// TwinCAT 3 PLC project mobject_core
// Title: mobject-core
// Company: mobject
// Author: mobject dev team
// ProjectVersion: 0.4.0
// ProgramVersion: 3.1.4024.0
// libraries:
//   Tc2_Standard, * (Beckhoff Automation GmbH)
//   Tc2_System, * (Beckhoff Automation GmbH)
//   Tc2_Utilities, * (Beckhoff Automation GmbH)
//   Tc3_DynamicMemory, * (Beckhoff Automation GmbH)
//   Tc3_JsonXml, * (Beckhoff Automation GmbH)
// project tree:
//   mobject-collections/Dictionary/ Dictionary.TcPOU
//   mobject-collections/Interfaces/Collections/Events/ I_CollectionChangedEvent.TcIO (not stored), I_CollectionDisposedEvent.TcIO (not stored)
//   mobject-collections/Interfaces/Collections/ I_Collection.TcIO, I_LinkedList.TcIO, I_List.TcIO (not stored), I_Queue.TcIO (not stored), I_Stack.TcIO
//   mobject-collections/Interfaces/Collections/Nodes/ I_CollectionNode.TcIO (not stored), I_LinkedListNode.TcIO (not stored), I_ListNode.TcIO (not stored)
//   mobject-collections/Interfaces/KeyValueCollections/Events/ I_KeyValueCollectionChangedEvent.TcIO (not stored), I_KeyValueCollectionDisposedEvent.TcIO (not stored)
//   mobject-collections/Interfaces/KeyValueCollections/ I_Dictionary.TcIO (not stored), I_KeyValueCollection.TcIO (not stored)
//   mobject-collections/Interfaces/KeyValueCollections/Nodes/ I_DictionaryTreeNode.TcIO, I_OrderedDictionaryTreeNode.TcIO
//   mobject-collections/LinkedList/ LinkedList.TcPOU
//   mobject-collections/List/ List.TcPOU
//   mobject-collections/OrderedDictionary/ OrderedDictionary.TcPOU
//   mobject-collections/Queue/ Queue.TcPOU (not stored)
//   mobject-collections/Stack/ Stack.TcPOU
//   mobject-collections/_Internal/Dictionary/Enumerator/ DictionaryForwardEnumerator.TcPOU
//   mobject-collections/_Internal/Dictionary/Node/ DictionaryTreeNode.TcPOU
//   mobject-collections/_Internal/Events/Collection/ CollectionChangedEvent.TcPOU (not stored), CollectionDisposedEvent.TcPOU (not stored), CollectionEvent.TcPOU (not stored)
//   mobject-collections/_Internal/Events/KeyValueCollection/ KeyValueCollectionChangedEvent.TcPOU, KeyValueCollectionDisposedEvent.TcPOU, KeyValueCollectionEvent.TcPOU
//   mobject-collections/_Internal/LinkedList/Enumerator/ LinkedListForwardEnumerator.TcPOU
//   mobject-collections/_Internal/LinkedList/Node/ LinkedListNode.TcPOU
//   mobject-collections/_Internal/List/Node/ ListNode.TcPOU
//   mobject-collections/_Internal/OrderedDictionary/Enumerator/ OrderedDictionaryForwardEnumerator.TcPOU (not stored)
//   mobject-collections/_Internal/OrderedDictionary/Node/ OrderedDictionaryTreeNode.TcPOU
//   mobject-commands/AsyncCommand/ AsyncCommand.TcPOU (not stored)
//   mobject-commands/AsyncCommand/Interface/ I_AsyncCommand.TcIO
//   mobject-commands/AsyncCommand/Runners/ SingleAsyncCommandRunner.TcPOU (not stored)
//   mobject-commands/Command/Interface/ I_Command.TcIO
//   mobject-commands/_Internal/AsyncCommandStateMachine/ AsyncCommandStateMachine.TcPOU, I_AsyncCommandStateControl.TcIO (not stored)
//   mobject-constants/ DatatypeLimits.TcGVL
//   mobject-converters/Converters/BOOL_TO_/ TryConvert_BOOL_TO_BOOL.TcPOU (not stored), TryConvert_BOOL_TO_BYTE.TcPOU, TryConvert_BOOL_TO_DATE.TcPOU, TryConvert_BOOL_TO_Destination.TcPOU, TryConvert_BOOL_TO_DINT.TcPOU, TryConvert_BOOL_TO_DT.TcPOU (not stored), TryConvert_BOOL_TO_DWORD.TcPOU (not stored), TryConvert_BOOL_TO_INT.TcPOU, TryConvert_BOOL_TO_LINT.TcPOU, TryConvert_BOOL_TO_LREAL.TcPOU (not stored), TryConvert_BOOL_TO_LWORD.TcPOU (not stored), TryConvert_BOOL_TO_REAL.TcPOU, TryConvert_BOOL_TO_SINT.TcPOU (not stored), TryConvert_BOOL_TO_STRING.TcPOU (not stored), TryConvert_BOOL_TO_TIME.TcPOU (not stored), TryConvert_BOOL_TO_TOD.TcPOU (not stored), TryConvert_BOOL_TO_UDINT.TcPOU, TryConvert_BOOL_TO_UINT.TcPOU, TryConvert_BOOL_TO_ULINT.TcPOU, TryConvert_BOOL_TO_USINT.TcPOU, TryConvert_BOOL_TO_WORD.TcPOU (not stored)
//   mobject-converters/Converters/BYTE_TO_/ TryConvert_BYTE_TO_BOOL.TcPOU, TryConvert_BYTE_TO_BYTE.TcPOU (not stored), TryConvert_BYTE_TO_DATE.TcPOU, TryConvert_BYTE_TO_Destination.TcPOU (not stored), TryConvert_BYTE_TO_DINT.TcPOU, TryConvert_BYTE_TO_DT.TcPOU (not stored), TryConvert_BYTE_TO_DWORD.TcPOU, TryConvert_BYTE_TO_INT.TcPOU, TryConvert_BYTE_TO_LINT.TcPOU (not stored), TryConvert_BYTE_TO_LREAL.TcPOU (not stored), TryConvert_BYTE_TO_LWORD.TcPOU (not stored), TryConvert_BYTE_TO_REAL.TcPOU, TryConvert_BYTE_TO_SINT.TcPOU, TryConvert_BYTE_TO_STRING.TcPOU, TryConvert_BYTE_TO_TIME.TcPOU, TryConvert_BYTE_TO_TOD.TcPOU, TryConvert_BYTE_TO_UDINT.TcPOU (not stored), TryConvert_BYTE_TO_UINT.TcPOU (not stored), TryConvert_BYTE_TO_ULINT.TcPOU, TryConvert_BYTE_TO_USINT.TcPOU, TryConvert_BYTE_TO_WORD.TcPOU
//   mobject-converters/Converters/DATE_TO_/ TryConvert_DATE_TO_BOOL.TcPOU (not stored), TryConvert_DATE_TO_BYTE.TcPOU (not stored), TryConvert_DATE_TO_DATE.TcPOU, TryConvert_DATE_TO_Destination.TcPOU (not stored), TryConvert_DATE_TO_DINT.TcPOU (not stored), TryConvert_DATE_TO_DT.TcPOU, TryConvert_DATE_TO_DWORD.TcPOU, TryConvert_DATE_TO_INT.TcPOU (not stored), TryConvert_DATE_TO_LINT.TcPOU (not stored), TryConvert_DATE_TO_LREAL.TcPOU, TryConvert_DATE_TO_LWORD.TcPOU, TryConvert_DATE_TO_REAL.TcPOU, TryConvert_DATE_TO_SINT.TcPOU (not stored), TryConvert_DATE_TO_STRING.TcPOU, TryConvert_DATE_TO_TIME.TcPOU (not stored), TryConvert_DATE_TO_TOD.TcPOU, TryConvert_DATE_TO_UDINT.TcPOU (not stored), TryConvert_DATE_TO_UINT.TcPOU, TryConvert_DATE_TO_ULINT.TcPOU, TryConvert_DATE_TO_USINT.TcPOU, TryConvert_DATE_TO_WORD.TcPOU
//   mobject-converters/Converters/DINT_TO_/ TryConvert_DINT_TO_BOOL.TcPOU (not stored), TryConvert_DINT_TO_BYTE.TcPOU (not stored), TryConvert_DINT_TO_DATE.TcPOU, TryConvert_DINT_TO_Destination.TcPOU, TryConvert_DINT_TO_DINT.TcPOU, TryConvert_DINT_TO_DT.TcPOU (not stored), TryConvert_DINT_TO_DWORD.TcPOU (not stored), TryConvert_DINT_TO_INT.TcPOU (not stored), TryConvert_DINT_TO_LINT.TcPOU (not stored), TryConvert_DINT_TO_LREAL.TcPOU (not stored), TryConvert_DINT_TO_LWORD.TcPOU, TryConvert_DINT_TO_REAL.TcPOU, TryConvert_DINT_TO_SINT.TcPOU, TryConvert_DINT_TO_STRING.TcPOU (not stored), TryConvert_DINT_TO_TIME.TcPOU (not stored), TryConvert_DINT_TO_TOD.TcPOU (not stored), TryConvert_DINT_TO_UDINT.TcPOU, TryConvert_DINT_TO_UINT.TcPOU (not stored), TryConvert_DINT_TO_ULINT.TcPOU, TryConvert_DINT_TO_USINT.TcPOU (not stored), TryConvert_DINT_TO_WORD.TcPOU (not stored)
//   mobject-converters/Converters/DT_TO_/ TryConvert_DT_TO_BOOL.TcPOU (not stored), TryConvert_DT_TO_BYTE.TcPOU (not stored), TryConvert_DT_TO_DATE.TcPOU, TryConvert_DT_TO_Destination.TcPOU, TryConvert_DT_TO_DINT.TcPOU (not stored), TryConvert_DT_TO_DT.TcPOU (not stored), TryConvert_DT_TO_DWORD.TcPOU (not stored), TryConvert_DT_TO_INT.TcPOU, TryConvert_DT_TO_LINT.TcPOU (not stored), TryConvert_DT_TO_LREAL.TcPOU, TryConvert_DT_TO_LWORD.TcPOU (not stored), TryConvert_DT_TO_REAL.TcPOU (not stored), TryConvert_DT_TO_SINT.TcPOU, TryConvert_DT_TO_STRING.TcPOU, TryConvert_DT_TO_TIME.TcPOU, TryConvert_DT_TO_TOD.TcPOU (not stored), TryConvert_DT_TO_UDINT.TcPOU, TryConvert_DT_TO_UINT.TcPOU (not stored), TryConvert_DT_TO_ULINT.TcPOU (not stored), TryConvert_DT_TO_USINT.TcPOU, TryConvert_DT_TO_WORD.TcPOU
//   mobject-converters/Converters/DWORD_TO_/ TryConvert_DWORD_TO_BOOL.TcPOU, TryConvert_DWORD_TO_BYTE.TcPOU (not stored), TryConvert_DWORD_TO_DATE.TcPOU (not stored), TryConvert_DWORD_TO_Destination.TcPOU (not stored), TryConvert_DWORD_TO_DINT.TcPOU (not stored), TryConvert_DWORD_TO_DT.TcPOU (not stored), TryConvert_DWORD_TO_DWORD.TcPOU (not stored), TryConvert_DWORD_TO_INT.TcPOU (not stored), TryConvert_DWORD_TO_LINT.TcPOU (not stored), TryConvert_DWORD_TO_LREAL.TcPOU, TryConvert_DWORD_TO_LWORD.TcPOU (not stored), TryConvert_DWORD_TO_REAL.TcPOU (not stored), TryConvert_DWORD_TO_SINT.TcPOU, TryConvert_DWORD_TO_STRING.TcPOU (not stored), TryConvert_DWORD_TO_TIME.TcPOU (not stored), TryConvert_DWORD_TO_TOD.TcPOU (not stored), TryConvert_DWORD_TO_UDINT.TcPOU, TryConvert_DWORD_TO_UINT.TcPOU, TryConvert_DWORD_TO_ULINT.TcPOU, TryConvert_DWORD_TO_USINT.TcPOU (not stored), TryConvert_DWORD_TO_WORD.TcPOU
//   mobject-converters/Converters/INT_TO_/ TryConvert_INT_TO_BOOL.TcPOU, TryConvert_INT_TO_BYTE.TcPOU, TryConvert_INT_TO_DATE.TcPOU (not stored), TryConvert_INT_TO_Destination.TcPOU, TryConvert_INT_TO_DINT.TcPOU, TryConvert_INT_TO_DT.TcPOU (not stored), TryConvert_INT_TO_DWORD.TcPOU, TryConvert_INT_TO_INT.TcPOU (not stored), TryConvert_INT_TO_LINT.TcPOU (not stored), TryConvert_INT_TO_LREAL.TcPOU, TryConvert_INT_TO_LWORD.TcPOU (not stored), TryConvert_INT_TO_REAL.TcPOU (not stored), TryConvert_INT_TO_SINT.TcPOU, TryConvert_INT_TO_STRING.TcPOU (not stored), TryConvert_INT_TO_TIME.TcPOU (not stored), TryConvert_INT_TO_TOD.TcPOU, TryConvert_INT_TO_UDINT.TcPOU (not stored), TryConvert_INT_TO_UINT.TcPOU, TryConvert_INT_TO_ULINT.TcPOU (not stored), TryConvert_INT_TO_USINT.TcPOU (not stored), TryConvert_INT_TO_WORD.TcPOU (not stored)
//   mobject-converters/Converters/LINT_TO_/ TryConvert_LINT_TO_BOOL.TcPOU (not stored), TryConvert_LINT_TO_BYTE.TcPOU (not stored), TryConvert_LINT_TO_DATE.TcPOU (not stored), TryConvert_LINT_TO_Destination.TcPOU, TryConvert_LINT_TO_DINT.TcPOU (not stored), TryConvert_LINT_TO_DT.TcPOU (not stored), TryConvert_LINT_TO_DWORD.TcPOU (not stored), TryConvert_LINT_TO_INT.TcPOU (not stored), TryConvert_LINT_TO_LINT.TcPOU (not stored), TryConvert_LINT_TO_LREAL.TcPOU (not stored), TryConvert_LINT_TO_LWORD.TcPOU, TryConvert_LINT_TO_REAL.TcPOU, TryConvert_LINT_TO_SINT.TcPOU, TryConvert_LINT_TO_STRING.TcPOU (not stored), TryConvert_LINT_TO_TIME.TcPOU (not stored), TryConvert_LINT_TO_TOD.TcPOU (not stored), TryConvert_LINT_TO_UDINT.TcPOU, TryConvert_LINT_TO_UINT.TcPOU (not stored), TryConvert_LINT_TO_ULINT.TcPOU (not stored), TryConvert_LINT_TO_USINT.TcPOU (not stored), TryConvert_LINT_TO_WORD.TcPOU
//   mobject-converters/Converters/LREAL_TO_/ TryConvert_LREAL_TO_BOOL.TcPOU (not stored), TryConvert_LREAL_TO_BYTE.TcPOU, TryConvert_LREAL_TO_DATE.TcPOU (not stored), TryConvert_LREAL_TO_Destination.TcPOU, TryConvert_LREAL_TO_DINT.TcPOU, TryConvert_LREAL_TO_DT.TcPOU (not stored), TryConvert_LREAL_TO_DWORD.TcPOU, TryConvert_LREAL_TO_INT.TcPOU (not stored), TryConvert_LREAL_TO_LINT.TcPOU, TryConvert_LREAL_TO_LREAL.TcPOU, TryConvert_LREAL_TO_LWORD.TcPOU, TryConvert_LREAL_TO_REAL.TcPOU, TryConvert_LREAL_TO_SINT.TcPOU, TryConvert_LREAL_TO_STRING.TcPOU (not stored), TryConvert_LREAL_TO_TIME.TcPOU, TryConvert_LREAL_TO_TOD.TcPOU, TryConvert_LREAL_TO_UDINT.TcPOU, TryConvert_LREAL_TO_UINT.TcPOU (not stored), TryConvert_LREAL_TO_ULINT.TcPOU (not stored), TryConvert_LREAL_TO_USINT.TcPOU (not stored), TryConvert_LREAL_TO_WORD.TcPOU (not stored)
//   mobject-converters/Converters/LWORD_TO_/ TryConvert_LWORD_TO_BOOL.TcPOU, TryConvert_LWORD_TO_BYTE.TcPOU (not stored), TryConvert_LWORD_TO_DATE.TcPOU (not stored), TryConvert_LWORD_TO_Destination.TcPOU, TryConvert_LWORD_TO_DINT.TcPOU, TryConvert_LWORD_TO_DT.TcPOU, TryConvert_LWORD_TO_DWORD.TcPOU (not stored), TryConvert_LWORD_TO_INT.TcPOU (not stored), TryConvert_LWORD_TO_LINT.TcPOU, TryConvert_LWORD_TO_LREAL.TcPOU, TryConvert_LWORD_TO_LWORD.TcPOU (not stored), TryConvert_LWORD_TO_REAL.TcPOU (not stored), TryConvert_LWORD_TO_SINT.TcPOU (not stored), TryConvert_LWORD_TO_STRING.TcPOU, TryConvert_LWORD_TO_TIME.TcPOU, TryConvert_LWORD_TO_TOD.TcPOU, TryConvert_LWORD_TO_UDINT.TcPOU, TryConvert_LWORD_TO_UINT.TcPOU, TryConvert_LWORD_TO_ULINT.TcPOU (not stored), TryConvert_LWORD_TO_USINT.TcPOU, TryConvert_LWORD_TO_WORD.TcPOU (not stored)
//   mobject-converters/Converters/REAL_TO_/ TryConvert_REAL_TO_BOOL.TcPOU, TryConvert_REAL_TO_BYTE.TcPOU, TryConvert_REAL_TO_DATE.TcPOU (not stored), TryConvert_REAL_TO_Destination.TcPOU, TryConvert_REAL_TO_DINT.TcPOU (not stored), TryConvert_REAL_TO_DT.TcPOU (not stored), TryConvert_REAL_TO_DWORD.TcPOU (not stored), TryConvert_REAL_TO_INT.TcPOU (not stored), TryConvert_REAL_TO_LINT.TcPOU (not stored), TryConvert_REAL_TO_LREAL.TcPOU, TryConvert_REAL_TO_LWORD.TcPOU, TryConvert_REAL_TO_REAL.TcPOU (not stored), TryConvert_REAL_TO_SINT.TcPOU (not stored), TryConvert_REAL_TO_STRING.TcPOU (not stored), TryConvert_REAL_TO_TIME.TcPOU (not stored), TryConvert_REAL_TO_TOD.TcPOU (not stored), TryConvert_REAL_TO_UDINT.TcPOU (not stored), TryConvert_REAL_TO_UINT.TcPOU (not stored), TryConvert_REAL_TO_ULINT.TcPOU (not stored), TryConvert_REAL_TO_USINT.TcPOU (not stored), TryConvert_REAL_TO_WORD.TcPOU (not stored)
//   mobject-converters/Converters/SINT_TO_/ TryConvert_SINT_TO_BOOL.TcPOU, TryConvert_SINT_TO_BYTE.TcPOU (not stored), TryConvert_SINT_TO_DATE.TcPOU, TryConvert_SINT_TO_Destination.TcPOU, TryConvert_SINT_TO_DINT.TcPOU, TryConvert_SINT_TO_DT.TcPOU (not stored), TryConvert_SINT_TO_DWORD.TcPOU, TryConvert_SINT_TO_INT.TcPOU (not stored), TryConvert_SINT_TO_LINT.TcPOU (not stored), TryConvert_SINT_TO_LREAL.TcPOU (not stored), TryConvert_SINT_TO_LWORD.TcPOU, TryConvert_SINT_TO_REAL.TcPOU, TryConvert_SINT_TO_SINT.TcPOU, TryConvert_SINT_TO_STRING.TcPOU, TryConvert_SINT_TO_TIME.TcPOU, TryConvert_SINT_TO_TOD.TcPOU, TryConvert_SINT_TO_UDINT.TcPOU (not stored), TryConvert_SINT_TO_UINT.TcPOU (not stored), TryConvert_SINT_TO_ULINT.TcPOU (not stored), TryConvert_SINT_TO_USINT.TcPOU, TryConvert_SINT_TO_WORD.TcPOU
//   mobject-converters/Converters/STRING_TO_/ TryConvert_STRING_TO_BOOL.TcPOU, TryConvert_STRING_TO_BYTE.TcPOU (not stored), TryConvert_STRING_TO_DATE.TcPOU (not stored), TryConvert_STRING_TO_Destination.TcPOU (not stored), TryConvert_STRING_TO_DINT.TcPOU (not stored), TryConvert_STRING_TO_DT.TcPOU, TryConvert_STRING_TO_DWORD.TcPOU (not stored), TryConvert_STRING_TO_INT.TcPOU, TryConvert_STRING_TO_LINT.TcPOU, TryConvert_STRING_TO_LREAL.TcPOU (not stored), TryConvert_STRING_TO_LWORD.TcPOU, TryConvert_STRING_TO_REAL.TcPOU (not stored), TryConvert_STRING_TO_SINT.TcPOU (not stored), TryConvert_STRING_TO_STRING.TcPOU (not stored), TryConvert_STRING_TO_TIME.TcPOU, TryConvert_STRING_TO_TOD.TcPOU (not stored), TryConvert_STRING_TO_UDINT.TcPOU, TryConvert_STRING_TO_UINT.TcPOU (not stored), TryConvert_STRING_TO_ULINT.TcPOU (not stored), TryConvert_STRING_TO_USINT.TcPOU (not stored), TryConvert_STRING_TO_WORD.TcPOU (not stored)
//   mobject-converters/Converters/TIME_TO_/ TryConvert_TIME_TO_BOOL.TcPOU (not stored), TryConvert_TIME_TO_BYTE.TcPOU (not stored), TryConvert_TIME_TO_DATE.TcPOU, TryConvert_TIME_TO_Destination.TcPOU, TryConvert_TIME_TO_DINT.TcPOU (not stored), TryConvert_TIME_TO_DT.TcPOU, TryConvert_TIME_TO_DWORD.TcPOU (not stored), TryConvert_TIME_TO_INT.TcPOU (not stored), TryConvert_TIME_TO_LINT.TcPOU, TryConvert_TIME_TO_LREAL.TcPOU, TryConvert_TIME_TO_LWORD.TcPOU (not stored), TryConvert_TIME_TO_REAL.TcPOU (not stored), TryConvert_TIME_TO_SINT.TcPOU (not stored), TryConvert_TIME_TO_STRING.TcPOU (not stored), TryConvert_TIME_TO_TIME.TcPOU (not stored), TryConvert_TIME_TO_TOD.TcPOU, TryConvert_TIME_TO_UDINT.TcPOU (not stored), TryConvert_TIME_TO_UINT.TcPOU, TryConvert_TIME_TO_ULINT.TcPOU, TryConvert_TIME_TO_USINT.TcPOU (not stored), TryConvert_TIME_TO_WORD.TcPOU (not stored)
//   mobject-converters/Converters/TOD_TO_/ TryConvert_TOD_TO_BOOL.TcPOU (not stored), TryConvert_TOD_TO_BYTE.TcPOU (not stored), TryConvert_TOD_TO_DATE.TcPOU, TryConvert_TOD_TO_Destination.TcPOU (not stored), TryConvert_TOD_TO_DINT.TcPOU, TryConvert_TOD_TO_DT.TcPOU, TryConvert_TOD_TO_DWORD.TcPOU, TryConvert_TOD_TO_INT.TcPOU (not stored), TryConvert_TOD_TO_LINT.TcPOU (not stored), TryConvert_TOD_TO_LREAL.TcPOU, TryConvert_TOD_TO_LWORD.TcPOU, TryConvert_TOD_TO_REAL.TcPOU (not stored), TryConvert_TOD_TO_SINT.TcPOU, TryConvert_TOD_TO_STRING.TcPOU, TryConvert_TOD_TO_TIME.TcPOU (not stored), TryConvert_TOD_TO_TOD.TcPOU, TryConvert_TOD_TO_UDINT.TcPOU, TryConvert_TOD_TO_UINT.TcPOU, TryConvert_TOD_TO_ULINT.TcPOU, TryConvert_TOD_TO_USINT.TcPOU (not stored), TryConvert_TOD_TO_WORD.TcPOU (not stored)
//   mobject-converters/Converters/ TryConvert_Source_TO_Destination.TcPOU
//   mobject-converters/Converters/UDINT_TO_/ TryConvert_UDINT_TO_BOOL.TcPOU (not stored), TryConvert_UDINT_TO_BYTE.TcPOU (not stored), TryConvert_UDINT_TO_DATE.TcPOU (not stored), TryConvert_UDINT_TO_Destination.TcPOU, TryConvert_UDINT_TO_DINT.TcPOU, TryConvert_UDINT_TO_DT.TcPOU, TryConvert_UDINT_TO_DWORD.TcPOU (not stored), TryConvert_UDINT_TO_INT.TcPOU (not stored), TryConvert_UDINT_TO_LINT.TcPOU, TryConvert_UDINT_TO_LREAL.TcPOU (not stored), TryConvert_UDINT_TO_LWORD.TcPOU (not stored), TryConvert_UDINT_TO_REAL.TcPOU (not stored), TryConvert_UDINT_TO_SINT.TcPOU, TryConvert_UDINT_TO_STRING.TcPOU (not stored), TryConvert_UDINT_TO_TIME.TcPOU, TryConvert_UDINT_TO_TOD.TcPOU, TryConvert_UDINT_TO_UDINT.TcPOU, TryConvert_UDINT_TO_UINT.TcPOU, TryConvert_UDINT_TO_ULINT.TcPOU, TryConvert_UDINT_TO_USINT.TcPOU (not stored), TryConvert_UDINT_TO_WORD.TcPOU (not stored)
//   mobject-converters/Converters/UINT_TO_/ TryConvert_UINT_TO_BOOL.TcPOU (not stored), TryConvert_UINT_TO_BYTE.TcPOU, TryConvert_UINT_TO_DATE.TcPOU (not stored), TryConvert_UINT_TO_Destination.TcPOU (not stored), TryConvert_UINT_TO_DINT.TcPOU, TryConvert_UINT_TO_DT.TcPOU, TryConvert_UINT_TO_DWORD.TcPOU (not stored), TryConvert_UINT_TO_INT.TcPOU (not stored), TryConvert_UINT_TO_LINT.TcPOU (not stored), TryConvert_UINT_TO_LREAL.TcPOU (not stored), TryConvert_UINT_TO_LWORD.TcPOU, TryConvert_UINT_TO_REAL.TcPOU (not stored), TryConvert_UINT_TO_SINT.TcPOU (not stored), TryConvert_UINT_TO_STRING.TcPOU, TryConvert_UINT_TO_TIME.TcPOU (not stored), TryConvert_UINT_TO_TOD.TcPOU (not stored), TryConvert_UINT_TO_UDINT.TcPOU (not stored), TryConvert_UINT_TO_UINT.TcPOU (not stored), TryConvert_UINT_TO_ULINT.TcPOU, TryConvert_UINT_TO_USINT.TcPOU, TryConvert_UINT_TO_WORD.TcPOU
//   mobject-converters/Converters/ULINT_TO_/ TryConvert_ULINT_TO_BOOL.TcPOU, TryConvert_ULINT_TO_BYTE.TcPOU (not stored), TryConvert_ULINT_TO_DATE.TcPOU (not stored), TryConvert_ULINT_TO_Destination.TcPOU (not stored), TryConvert_ULINT_TO_DINT.TcPOU, TryConvert_ULINT_TO_DT.TcPOU, TryConvert_ULINT_TO_DWORD.TcPOU (not stored), TryConvert_ULINT_TO_INT.TcPOU (not stored), TryConvert_ULINT_TO_LINT.TcPOU (not stored), TryConvert_ULINT_TO_LREAL.TcPOU (not stored), TryConvert_ULINT_TO_LWORD.TcPOU, TryConvert_ULINT_TO_REAL.TcPOU (not stored), TryConvert_ULINT_TO_SINT.TcPOU, TryConvert_ULINT_TO_STRING.TcPOU, TryConvert_ULINT_TO_TIME.TcPOU (not stored), TryConvert_ULINT_TO_TOD.TcPOU (not stored), TryConvert_ULINT_TO_UDINT.TcPOU, TryConvert_ULINT_TO_UINT.TcPOU (not stored), TryConvert_ULINT_TO_ULINT.TcPOU (not stored), TryConvert_ULINT_TO_USINT.TcPOU, TryConvert_ULINT_TO_WORD.TcPOU (not stored)
//   mobject-converters/Converters/USINT_TO_/ TryConvert_USINT_TO_BOOL.TcPOU, TryConvert_USINT_TO_BYTE.TcPOU, TryConvert_USINT_TO_DATE.TcPOU (not stored), TryConvert_USINT_TO_Destination.TcPOU (not stored), TryConvert_USINT_TO_DINT.TcPOU, TryConvert_USINT_TO_DT.TcPOU, TryConvert_USINT_TO_DWORD.TcPOU (not stored), TryConvert_USINT_TO_INT.TcPOU, TryConvert_USINT_TO_LINT.TcPOU (not stored), TryConvert_USINT_TO_LREAL.TcPOU (not stored), TryConvert_USINT_TO_LWORD.TcPOU, TryConvert_USINT_TO_REAL.TcPOU (not stored), TryConvert_USINT_TO_SINT.TcPOU (not stored), TryConvert_USINT_TO_STRING.TcPOU (not stored), TryConvert_USINT_TO_TIME.TcPOU (not stored), TryConvert_USINT_TO_TOD.TcPOU, TryConvert_USINT_TO_UDINT.TcPOU (not stored), TryConvert_USINT_TO_UINT.TcPOU, TryConvert_USINT_TO_ULINT.TcPOU, TryConvert_USINT_TO_USINT.TcPOU (not stored), TryConvert_USINT_TO_WORD.TcPOU (not stored)
//   mobject-converters/Converters/WORD_TO_/ TryConvert_WORD_TO_BOOL.TcPOU, TryConvert_WORD_TO_BYTE.TcPOU (not stored), TryConvert_WORD_TO_DATE.TcPOU (not stored), TryConvert_WORD_TO_Destination.TcPOU (not stored), TryConvert_WORD_TO_DINT.TcPOU (not stored), TryConvert_WORD_TO_DT.TcPOU, TryConvert_WORD_TO_DWORD.TcPOU (not stored), TryConvert_WORD_TO_INT.TcPOU (not stored), TryConvert_WORD_TO_LINT.TcPOU, TryConvert_WORD_TO_LREAL.TcPOU (not stored), TryConvert_WORD_TO_LWORD.TcPOU, TryConvert_WORD_TO_REAL.TcPOU, TryConvert_WORD_TO_SINT.TcPOU, TryConvert_WORD_TO_STRING.TcPOU (not stored), TryConvert_WORD_TO_TIME.TcPOU, TryConvert_WORD_TO_TOD.TcPOU (not stored), TryConvert_WORD_TO_UDINT.TcPOU (not stored), TryConvert_WORD_TO_UINT.TcPOU (not stored), TryConvert_WORD_TO_ULINT.TcPOU, TryConvert_WORD_TO_USINT.TcPOU, TryConvert_WORD_TO_WORD.TcPOU (not stored)
//   mobject-datatypes/DatatypeOperations/Collection/ DatatypeOperations.TcPOU
//   mobject-datatypes/DatatypeOperations/Interface/ I_DatatypeOperation.TcIO
//   mobject-datatypes/DatatypeOperations/ MemCopyOperation.TcPOU, SafeMemCopyOperation.TcPOU, WriteBitToBoolOperation.TcPOU (not stored), WriteBoolToBitOperation.TcPOU (not stored)
//   mobject-datatypes/Datatypes/Base/ Datatypes.TcPOU
//   mobject-datatypes/Datatypes/Events/ I_AliasDatatypeAddedEvent.TcIO, I_DatatypeAddedEvent.TcIO (not stored), I_EnumDatatypeAddedEvent.TcIO (not stored), I_InterfaceDatatypeAddedEvent.TcIO, I_StructuredDatatypeAddedEvent.TcIO, I_ArrayDatatypeAddedEvent.TcIO
//   mobject-datatypes/Datatypes/Interface/ I_Datatypes.TcIO
//   mobject-datatypes/DatatypeVisitor/ I_DatatypeVisitor.TcIO (not stored)
//   mobject-datatypes/Functions/ GetByteOffset.TcPOU
//   mobject-datatypes/Primitive/ _BIT.TcPOU, _BOOL.TcPOU, _BYTE.TcPOU, _DINT.TcPOU, _DT.TcPOU, _DWORD.TcPOU, _INT.TcPOU, _LINT.TcPOU, _LREAL.TcPOU, _LWORD.TcPOU, _REAL.TcPOU, _SINT.TcPOU, _STRING.TcPOU, _TIME_OF_DAY.TcPOU, _TOD.TcPOU, _UDINT.TcPOU, _PVOID.TcPOU (excluded from build), _UINT.TcPOU, _ULINT.TcPOU, _USINT.TcPOU, _WORD.TcPOU
//   mobject-datatypes/_Internal/Datatype/ AliasDatatypeBase.TcPOU, ArrayDatatypeBase_2D.TcPOU, ArrayDatatypeBase_3D.TcPOU (not stored), DatatypeBase.TcPOU, EnumDatatypeBase.TcPOU, InterfaceDatatypeBase.TcPOU, NumericDatatypeBase.TcPOU, StructuredDatatypeBase.TcPOU, ArrayDatatypeBase_1D.TcPOU, UserDefinedDatatypeBase.TcPOU
//   mobject-datatypes/_Internal/Datatype/Interface/ I_AliasDatatype.TcIO, I_ArrayDatatype_1D.TcIO (not stored), I_ArrayDatatype_2D.TcIO, I_ArrayDatatype_3D.TcIO (not stored), I_BitDatatype.TcIO, I_Datatype.TcIO, I_EnumDatatype.TcIO (not stored), I_InterfaceDatatype.TcIO (not stored), I_NumericDatatype.TcIO, I_StructuredDatatype.TcIO (not stored), I_ArrayDatatype.TcIO, I_UserDefinedDatatype.TcIO (not stored)
//   mobject-datatypes/_Internal/Errors/ UnknownEnumerationError.TcPOU
//   mobject-datatypes/_Internal/Events/ AliasDatatypeAddedEvent.TcPOU, DatatypeAddedEvent.TcPOU (not stored), EnumDatatypeAddedEvent.TcPOU, InterfaceDatatypeAddedEvent.TcPOU (not stored), StructuredDatatypeAddedEvent.TcPOU (not stored), ArrayDatatypeAddedEvent.TcPOU
//   mobject-datatypes/_Internal/StructureMembers/Host/ StructureMemberHost.TcPOU
//   mobject-datatypes/_Internal/StructureMembers/Interface/ I_HostStructureMembers.TcIO (not stored), I_StructureMembers.TcIO
//   mobject-deserialization/DeserializationFeedback/ DeserializerFeedback.TcPOU (not stored)
//   mobject-deserialization/Errors/CustomError/ CustomDeserializationFailedError.TcPOU
//   mobject-deserialization/Errors/ DeserializationErrorFactory.TcPOU
//   mobject-deserialization/Errors/IncorrectType/ IncorrectKeyTypeDeserializationError.TcPOU (not stored), IncorrectTypeDeserializationError.TcPOU (not stored)
//   mobject-deserialization/Errors/Invalid Index/ InvalidArrayIndexDeserializationError.TcPOU
//   mobject-deserialization/Errors/Invalid Key/ InvalidKeyDeserializationError.TcPOU
//   mobject-deserialization/Errors/Missing Key/ MissingKeyDeserializationError.TcPOU (not stored)
//   mobject-deserialization/GarbageCollector/ DeserializerGarbageCollector.TcPOU (not stored), I_DeserializerGarbageCollector.TcIO
//   mobject-deserialization/Interfaces/ I_Deserializable.TcIO, I_Deserializer.TcIO, I_DeserializerArrayForwardEnumerator.TcIO (not stored), I_DeserializerFeedback.TcIO (not stored), I_DeserializerObjectForwardEnumerator.TcIO (not stored)
//   mobject-errors/Errors/ Error.TcPOU, NullError.TcPOU (not stored)
//   mobject-errors/Interfaces/ I_Error.TcIO (not stored), I_ErrorVisitor.TcIO (not stored)
//   mobject-events/EventEmitter/ EventEmitter.TcPOU
//   mobject-events/Interfaces/ I_Event.TcIO (not stored), I_EventEmitter.TcIO, I_EventHandler.TcIO, I_EventTarget.TcIO
//   mobject-events/_Internal/EventHandlerItem/ EventHandlerItem.TcPOU, EventHandlerItemOnceOnly.TcPOU (not stored), I_EventHandlerItem.TcIO (not stored)
//   mobject-disposable/Disposable/ Disposable.TcPOU (not stored)
//   mobject-disposable/Interfaces/ I_Disposable.TcIO (not stored)
//   mobject-enumerable/Interfaces/Enumerators/ I_ForwardEnumerator.TcIO (not stored), I_KeyValueForwardEnumerator.TcIO
//   mobject-enumerable/Interfaces/ I_Enumerable.TcIO (not stored), I_KeyValueEnumerable.TcIO (not stored)
//   mobject-json/JsonDeserializer/Events/ I_JsonDeserializerChangedEvent.TcIO, I_JsonDeserializerDisposedEvent.TcIO (not stored)
//   mobject-json/JsonDeserializer/ I_JsonDeserializer.TcIO (not stored), JsonDeserializer.TcPOU
//   mobject-json/JsonDomParser/ JsonDomParser.TcPOU (not stored)
//   mobject-json/JsonSerializer/ JsonSerializer.TcPOU (not stored)
//   mobject-json/_Internal/Events/ JsonDeserializerChangedEvent.TcPOU (not stored), JsonDeserializerDisposedEvent.TcPOU, JsonDeserializerEvent.TcPOU (not stored)
//   mobject-json/_Internal/JsonDeserializerForwardEnumerator/ JsonDeserializerArrayForwardEnumerator.TcPOU, JsonDeserializerNullArrayForwardEnumerator.TcPOU (not stored), JsonDeserializerNullObjectForwardEnumerator.TcPOU, JsonDeserializerObjectForwardEnumerator.TcPOU
//   mobject-json/_Internal/JsonDeserializerNode/ JsonDeserializerNode.TcPOU, JsonDeserializerNullNode.TcPOU
//   mobject-json/_Internal/JsonPathSyntaxParser/ JsonPathSyntaxParser.TcPOU (not stored)
//   mobject-json/_Internal/JsonPathVisitor/ I_JsonPathVisitor.TcIO, JsonDomCreator.TcPOU (not stored), JsonDomNavigator.TcPOU
//   mobject-serialization/Interfaces/ I_Serializable.TcIO (not stored), I_Serializer.TcIO (not stored)

// ---- mobject-constants/DatatypeLimits.TcGVL
{attribute 'qualified_only'}
VAR_GLOBAL CONSTANT
                
	// Boolean
	BOOL_MIN_VALUE : BOOL := FALSE;
	BOOL_MAX_VALUE : BOOL := TRUE;
	
	// Integer Datatypes
	BYTE_MIN_VALUE : BYTE := BYTE#0;
	BYTE_MAX_VALUE : BYTE := BYTE#255;
	WORD_MIN_VALUE : WORD := WORD#0;
	WORD_MAX_VALUE : WORD := WORD#65535;
	DWORD_MIN_VALUE : DWORD := DWORD#0;
	DWORD_MAX_VALUE : DWORD := DWORD#4294967295;
	LWORD_MIN_VALUE : LWORD := LWORD#0;
	LWORD_MAX_VALUE : LWORD := LWORD#18446744073709551615;
	SINT_MIN_VALUE : SINT := SINT#-128;
	SINT_MAX_VALUE : SINT := SINT#127;
	USINT_MIN_VALUE : USINT := USINT#0;
	USINT_MAX_VALUE : USINT := USINT#255;
	INT_MIN_VALUE : INT := INT#-32768;
	INT_MAX_VALUE : INT := INT#32767;
	UINT_MIN_VALUE : UINT := UINT#0;
	UINT_MAX_VALUE : UINT := UINT#65535;
	DINT_MIN_VALUE : DINT := DINT#-2147483648;
	DINT_MAX_VALUE : DINT := DINT#2147483647;
	UDINT_MIN_VALUE : UDINT := UDINT#0;
	UDINT_MAX_VALUE : UDINT := UDINT#4294967295;
	LINT_MIN_VALUE : LINT := LINT#-9223372036854775808;
	LINT_MAX_VALUE : LINT := LINT#9223372036854775807;
	ULINT_MIN_VALUE : ULINT := ULINT#0;
	ULINT_MAX_VALUE : ULINT := ULINT#18446744073709551615;
	
	// Floating-point types
	REAL_MAX_VALUE : REAL := REAL#3.402823E+38; // Largest positive REAL number
	REAL_MIN_VALUE : REAL := REAL#-3.402823E+38; // Largest negative REAL number
	REAL_POSITIVE_MIN_VALUE : REAL := REAL#1.0E-44; // Smallest positive REAL number
	REAL_NEGATIVE_MIN_VALUE : REAL := REAL#-1.0E-44; // Smallest negative REAL number
	LREAL_MAX_VALUE : LREAL := LREAL#1.7976931348623157E+308; // Largest positive LREAL number
	LREAL_MIN_VALUE : LREAL := LREAL#-1.7976931348623157E+308; // Largest negative LREAL number
	LREAL_POSITIVE_MIN_VALUE : LREAL := LREAL#4.94065645841247E-324; // Smallest positive LREAL number
	LREAL_NEGATIVE_MIN_VALUE : LREAL := LREAL#-4.94065645841247E-324; // Smallest negative LREAL number
	
	// Time Datatypes
	TIME_MIN_VALUE : TIME := T#0MS;
	TIME_MAX_VALUE : TIME := T#49D17H2M47S295MS;
	
	// Date
	DATE_MIN_VALUE : DATE := DATE#1970-1-1;
	DATE_MAX_VALUE : DATE := DATE#2106-2-7;
	DT_MIN_VALUE : DATE_AND_TIME := DATE_AND_TIME#1970-1-1-0:0:0;
	DT_MAX_VALUE : DATE_AND_TIME := DATE_AND_TIME#2106-02-07-06:28:15;
	TOD_MIN_VALUE : TIME_OF_DAY := TIME_OF_DAY#0:0:0;
	TOD_MAX_VALUE : TIME_OF_DAY := TIME_OF_DAY#23:59:59.999;
	
	// -----------------------------------------------------------------------------
	
	// Limits of BYTE used for conversions
	MAX_VALUE_OF_BYTE_WHICH_CAN_BE_HELD_IN_A_SINT : BYTE := BYTE#127;
	
	// Limits of WORD used for conversions
	MAX_VALUE_OF_WORD_WHICH_CAN_BE_HELD_IN_A_BYTE : WORD := WORD#255;
	MAX_VALUE_OF_WORD_WHICH_CAN_BE_HELD_IN_A_SINT : WORD := WORD#127;
	MAX_VALUE_OF_WORD_WHICH_CAN_BE_HELD_IN_A_INT : WORD := WORD#32767;
	MAX_VALUE_OF_WORD_WHICH_CAN_BE_HELD_IN_A_USINT : WORD := WORD#255;
	
	// Limits of DWORD used for conversions
	MAX_VALUE_OF_DWORD_WHICH_CAN_BE_HELD_IN_A_BYTE : DWORD := DWORD#255;
	MAX_VALUE_OF_DWORD_WHICH_CAN_BE_HELD_IN_A_WORD : DWORD := DWORD#65535;
	MAX_VALUE_OF_DWORD_WHICH_CAN_BE_HELD_IN_A_SINT : DWORD := DWORD#127;
	MAX_VALUE_OF_DWORD_WHICH_CAN_BE_HELD_IN_A_INT : DWORD := DWORD#32767;
	MAX_VALUE_OF_DWORD_WHICH_CAN_BE_HELD_IN_A_DINT : DWORD := DWORD#2147483647;
	MAX_VALUE_OF_DWORD_WHICH_CAN_BE_HELD_IN_A_USINT : DWORD := DWORD#255;
	MAX_VALUE_OF_DWORD_WHICH_CAN_BE_HELD_IN_A_UINT : DWORD := DWORD#65535;
	MAX_VALUE_OF_DWORD_WHICH_CAN_BE_HELD_IN_A_TOD : DWORD := DWORD#86399999;
	
	// Limits of LWORD used for conversions
	MAX_VALUE_OF_LWORD_WHICH_CAN_BE_HELD_IN_A_BYTE : LWORD := LWORD#255;
	MAX_VALUE_OF_LWORD_WHICH_CAN_BE_HELD_IN_A_WORD : LWORD := LWORD#65535;
	MAX_VALUE_OF_LWORD_WHICH_CAN_BE_HELD_IN_A_DWORD : LWORD := LWORD#4294967295;
	MAX_VALUE_OF_LWORD_WHICH_CAN_BE_HELD_IN_A_SINT : LWORD := LWORD#127;
	MAX_VALUE_OF_LWORD_WHICH_CAN_BE_HELD_IN_A_INT : LWORD := LWORD#32767;
	MAX_VALUE_OF_LWORD_WHICH_CAN_BE_HELD_IN_A_DINT : LWORD := LWORD#2147483647;
	MAX_VALUE_OF_LWORD_WHICH_CAN_BE_HELD_IN_A_LINT : LWORD := LWORD#9223372036854775807;
	MAX_VALUE_OF_LWORD_WHICH_CAN_BE_HELD_IN_A_USINT : LWORD := LWORD#255;
	MAX_VALUE_OF_LWORD_WHICH_CAN_BE_HELD_IN_A_UINT : LWORD := LWORD#65535;
	MAX_VALUE_OF_LWORD_WHICH_CAN_BE_HELD_IN_A_UDINT : LWORD := LWORD#4294967295;
	MAX_VALUE_OF_LWORD_WHICH_CAN_BE_HELD_IN_A_TIME : LWORD := LWORD#4294967295;
	MAX_VALUE_OF_LWORD_WHICH_CAN_BE_HELD_IN_A_TOD : LWORD := LWORD#86399999;
	MAX_VALUE_OF_LWORD_WHICH_CAN_BE_HELD_IN_A_DATE : LWORD := LWORD#4294967295;
	MAX_VALUE_OF_LWORD_WHICH_CAN_BE_HELD_IN_A_DT : LWORD := LWORD#4294967295;
	
	// Limits of SINT used for conversions
	MIN_VALUE_OF_SINT_WHICH_CAN_BE_HELD_IN_A_BYTE : SINT := SINT#0;
	MIN_VALUE_OF_SINT_WHICH_CAN_BE_HELD_IN_A_WORD : SINT := SINT#0;
	MIN_VALUE_OF_SINT_WHICH_CAN_BE_HELD_IN_A_DWORD : SINT := SINT#0;
	MIN_VALUE_OF_SINT_WHICH_CAN_BE_HELD_IN_A_LWORD : SINT := SINT#0;
	MIN_VALUE_OF_SINT_WHICH_CAN_BE_HELD_IN_A_USINT : SINT := SINT#0;
	MIN_VALUE_OF_SINT_WHICH_CAN_BE_HELD_IN_A_UINT : SINT := SINT#0;
	MIN_VALUE_OF_SINT_WHICH_CAN_BE_HELD_IN_A_UDINT : SINT := SINT#0;
	MIN_VALUE_OF_SINT_WHICH_CAN_BE_HELD_IN_A_ULINT : SINT := SINT#0;
	MIN_VALUE_OF_SINT_WHICH_CAN_BE_HELD_IN_A_TIME : SINT := SINT#0;
	MIN_VALUE_OF_SINT_WHICH_CAN_BE_HELD_IN_A_TOD : SINT := SINT#0;
	MIN_VALUE_OF_SINT_WHICH_CAN_BE_HELD_IN_A_DATE : SINT := SINT#0;
	MIN_VALUE_OF_SINT_WHICH_CAN_BE_HELD_IN_A_DT : SINT := SINT#0;
	
	// Limits of INT used for conversions
	MIN_VALUE_OF_INT_WHICH_CAN_BE_HELD_IN_A_BYTE : INT := INT#0;
	MAX_VALUE_OF_INT_WHICH_CAN_BE_HELD_IN_A_BYTE : INT := INT#255;
	MIN_VALUE_OF_INT_WHICH_CAN_BE_HELD_IN_A_WORD : INT := INT#0;
	MIN_VALUE_OF_INT_WHICH_CAN_BE_HELD_IN_A_DWORD : INT := INT#0;
	MIN_VALUE_OF_INT_WHICH_CAN_BE_HELD_IN_A_LWORD : INT := INT#0;
	MIN_VALUE_OF_INT_WHICH_CAN_BE_HELD_IN_A_SINT : INT := INT#-128;
	MAX_VALUE_OF_INT_WHICH_CAN_BE_HELD_IN_A_SINT : INT := INT#127;
	MIN_VALUE_OF_INT_WHICH_CAN_BE_HELD_IN_A_USINT : INT := INT#0;
	MAX_VALUE_OF_INT_WHICH_CAN_BE_HELD_IN_A_USINT : INT := INT#255;
	MIN_VALUE_OF_INT_WHICH_CAN_BE_HELD_IN_A_UINT : INT := INT#0;
	MIN_VALUE_OF_INT_WHICH_CAN_BE_HELD_IN_A_UDINT : INT := INT#0;
	MIN_VALUE_OF_INT_WHICH_CAN_BE_HELD_IN_A_ULINT : INT := INT#0;
	MIN_VALUE_OF_INT_WHICH_CAN_BE_HELD_IN_A_TIME : INT := INT#0;
	MIN_VALUE_OF_INT_WHICH_CAN_BE_HELD_IN_A_TOD : INT := INT#0;
	MIN_VALUE_OF_INT_WHICH_CAN_BE_HELD_IN_A_DATE : INT := INT#0;
	MIN_VALUE_OF_INT_WHICH_CAN_BE_HELD_IN_A_DT : INT := INT#0;
	
	// Limits of DINT used for conversions
	MIN_VALUE_OF_DINT_WHICH_CAN_BE_HELD_IN_A_BYTE : DINT := DINT#0;
	MAX_VALUE_OF_DINT_WHICH_CAN_BE_HELD_IN_A_BYTE : DINT := DINT#255;
	MIN_VALUE_OF_DINT_WHICH_CAN_BE_HELD_IN_A_WORD : DINT := DINT#0;
	MAX_VALUE_OF_DINT_WHICH_CAN_BE_HELD_IN_A_WORD : DINT := DINT#65535;
	MIN_VALUE_OF_DINT_WHICH_CAN_BE_HELD_IN_A_DWORD : DINT := DINT#0;
	MIN_VALUE_OF_DINT_WHICH_CAN_BE_HELD_IN_A_LWORD : DINT := DINT#0;
	MIN_VALUE_OF_DINT_WHICH_CAN_BE_HELD_IN_A_SINT : DINT := DINT#-128;
	MAX_VALUE_OF_DINT_WHICH_CAN_BE_HELD_IN_A_SINT : DINT := DINT#127;
	MIN_VALUE_OF_DINT_WHICH_CAN_BE_HELD_IN_A_INT : DINT := DINT#-32768;
	MAX_VALUE_OF_DINT_WHICH_CAN_BE_HELD_IN_A_INT : DINT := DINT#32767;
	MIN_VALUE_OF_DINT_WHICH_CAN_BE_HELD_IN_A_USINT : DINT := DINT#0;
	MAX_VALUE_OF_DINT_WHICH_CAN_BE_HELD_IN_A_USINT : DINT := DINT#255;
	MIN_VALUE_OF_DINT_WHICH_CAN_BE_HELD_IN_A_UINT : DINT := DINT#0;
	MAX_VALUE_OF_DINT_WHICH_CAN_BE_HELD_IN_A_UINT : DINT := DINT#65535;
	MIN_VALUE_OF_DINT_WHICH_CAN_BE_HELD_IN_A_UDINT : DINT := DINT#0;
	MIN_VALUE_OF_DINT_WHICH_CAN_BE_HELD_IN_A_ULINT : DINT := DINT#0;
	MIN_VALUE_OF_DINT_WHICH_CAN_BE_HELD_IN_A_TIME : DINT := DINT#0;
	MIN_VALUE_OF_DINT_WHICH_CAN_BE_HELD_IN_A_TOD : DINT := DINT#0;
	MAX_VALUE_OF_DINT_WHICH_CAN_BE_HELD_IN_A_TOD : DINT := DINT#86399999;
	MIN_VALUE_OF_DINT_WHICH_CAN_BE_HELD_IN_A_DATE : DINT := DINT#0;
	MIN_VALUE_OF_DINT_WHICH_CAN_BE_HELD_IN_A_DT : DINT := DINT#0;
	
	// Limits of LINT used for conversions
	MIN_VALUE_OF_LINT_WHICH_CAN_BE_HELD_IN_A_BYTE : LINT := LINT#0;
	MAX_VALUE_OF_LINT_WHICH_CAN_BE_HELD_IN_A_BYTE : LINT := LINT#255;
	MIN_VALUE_OF_LINT_WHICH_CAN_BE_HELD_IN_A_WORD : LINT := LINT#0;
	MAX_VALUE_OF_LINT_WHICH_CAN_BE_HELD_IN_A_WORD : LINT := LINT#65535;
	MIN_VALUE_OF_LINT_WHICH_CAN_BE_HELD_IN_A_DWORD : LINT := LINT#0;
	MAX_VALUE_OF_LINT_WHICH_CAN_BE_HELD_IN_A_DWORD : LINT := LINT#4294967295;
	MIN_VALUE_OF_LINT_WHICH_CAN_BE_HELD_IN_A_LWORD : LINT := LINT#0;
	MIN_VALUE_OF_LINT_WHICH_CAN_BE_HELD_IN_A_SINT : LINT := LINT#-128;
	MAX_VALUE_OF_LINT_WHICH_CAN_BE_HELD_IN_A_SINT : LINT := LINT#127;
	MIN_VALUE_OF_LINT_WHICH_CAN_BE_HELD_IN_A_INT : LINT := LINT#-32768;
	MAX_VALUE_OF_LINT_WHICH_CAN_BE_HELD_IN_A_INT : LINT := LINT#32767;
	MIN_VALUE_OF_LINT_WHICH_CAN_BE_HELD_IN_A_DINT : LINT := LINT#-2147483648;
	MAX_VALUE_OF_LINT_WHICH_CAN_BE_HELD_IN_A_DINT : LINT := LINT#2147483647;
	MIN_VALUE_OF_LINT_WHICH_CAN_BE_HELD_IN_A_USINT : LINT := LINT#0;
	MAX_VALUE_OF_LINT_WHICH_CAN_BE_HELD_IN_A_USINT : LINT := LINT#255;
	MIN_VALUE_OF_LINT_WHICH_CAN_BE_HELD_IN_A_UINT : LINT := LINT#0;
	MAX_VALUE_OF_LINT_WHICH_CAN_BE_HELD_IN_A_UINT : LINT := LINT#65535;
	MIN_VALUE_OF_LINT_WHICH_CAN_BE_HELD_IN_A_UDINT : LINT := LINT#0;
	MAX_VALUE_OF_LINT_WHICH_CAN_BE_HELD_IN_A_UDINT : LINT := LINT#4294967295;
	MIN_VALUE_OF_LINT_WHICH_CAN_BE_HELD_IN_A_ULINT : LINT := LINT#0;
	MIN_VALUE_OF_LINT_WHICH_CAN_BE_HELD_IN_A_TIME : LINT := LINT#0;
	MAX_VALUE_OF_LINT_WHICH_CAN_BE_HELD_IN_A_TIME : LINT := LINT#4294967295;
	MIN_VALUE_OF_LINT_WHICH_CAN_BE_HELD_IN_A_TOD : LINT := LINT#0;
	MAX_VALUE_OF_LINT_WHICH_CAN_BE_HELD_IN_A_TOD : LINT := LINT#86399999;
	MIN_VALUE_OF_LINT_WHICH_CAN_BE_HELD_IN_A_DATE : LINT := LINT#0;
	MAX_VALUE_OF_LINT_WHICH_CAN_BE_HELD_IN_A_DATE : LINT := LINT#4294944000;
	MIN_VALUE_OF_LINT_WHICH_CAN_BE_HELD_IN_A_DT : LINT := LINT#0;
	MAX_VALUE_OF_LINT_WHICH_CAN_BE_HELD_IN_A_DT : LINT := LINT#4294967295;
	
	// Limits of USINT used for conversions
	MAX_VALUE_OF_USINT_WHICH_CAN_BE_HELD_IN_A_SINT : USINT := USINT#127;
	
	// Limits of UINT used for conversions
	MAX_VALUE_OF_UINT_WHICH_CAN_BE_HELD_IN_A_BYTE : UINT := UINT#255;
	MAX_VALUE_OF_UINT_WHICH_CAN_BE_HELD_IN_A_SINT : UINT := UINT#127;
	MAX_VALUE_OF_UINT_WHICH_CAN_BE_HELD_IN_A_INT : UINT := UINT#32767;
	MAX_VALUE_OF_UINT_WHICH_CAN_BE_HELD_IN_A_USINT : UINT := UINT#255;
	
	// Limits of UDINT used for conversions
	MAX_VALUE_OF_UDINT_WHICH_CAN_BE_HELD_IN_A_BYTE : UDINT := UDINT#255;
	MAX_VALUE_OF_UDINT_WHICH_CAN_BE_HELD_IN_A_WORD : UDINT := UDINT#65535;
	MAX_VALUE_OF_UDINT_WHICH_CAN_BE_HELD_IN_A_SINT : UDINT := UDINT#127;
	MAX_VALUE_OF_UDINT_WHICH_CAN_BE_HELD_IN_A_INT : UDINT := UDINT#32767;
	MAX_VALUE_OF_UDINT_WHICH_CAN_BE_HELD_IN_A_DINT : UDINT := UDINT#2147483647;
	MAX_VALUE_OF_UDINT_WHICH_CAN_BE_HELD_IN_A_USINT : UDINT := UDINT#255;
	MAX_VALUE_OF_UDINT_WHICH_CAN_BE_HELD_IN_A_UINT : UDINT := UDINT#65535;
	MAX_VALUE_OF_UDINT_WHICH_CAN_BE_HELD_IN_A_TOD : UDINT := UDINT#86399999;
	
	// Limits of ULINT used for conversions
	MAX_VALUE_OF_ULINT_WHICH_CAN_BE_HELD_IN_A_BYTE : ULINT := ULINT#255;
	MAX_VALUE_OF_ULINT_WHICH_CAN_BE_HELD_IN_A_WORD : ULINT := ULINT#65535;
	MAX_VALUE_OF_ULINT_WHICH_CAN_BE_HELD_IN_A_DWORD : ULINT := ULINT#4294967295;
	MAX_VALUE_OF_ULINT_WHICH_CAN_BE_HELD_IN_A_SINT : ULINT := ULINT#127;
	MAX_VALUE_OF_ULINT_WHICH_CAN_BE_HELD_IN_A_INT : ULINT := ULINT#32767;
	MAX_VALUE_OF_ULINT_WHICH_CAN_BE_HELD_IN_A_DINT : ULINT := ULINT#2147483647;
	MAX_VALUE_OF_ULINT_WHICH_CAN_BE_HELD_IN_A_LINT : ULINT := ULINT#9223372036854775807;
	MAX_VALUE_OF_ULINT_WHICH_CAN_BE_HELD_IN_A_USINT : ULINT := ULINT#255;
	MAX_VALUE_OF_ULINT_WHICH_CAN_BE_HELD_IN_A_UINT : ULINT := ULINT#65535;
	MAX_VALUE_OF_ULINT_WHICH_CAN_BE_HELD_IN_A_UDINT : ULINT := ULINT#4294967295;
	MAX_VALUE_OF_ULINT_WHICH_CAN_BE_HELD_IN_A_TIME : ULINT := ULINT#4294967295;
	MAX_VALUE_OF_ULINT_WHICH_CAN_BE_HELD_IN_A_TOD : ULINT := ULINT#86399999;
	MAX_VALUE_OF_ULINT_WHICH_CAN_BE_HELD_IN_A_DATE : ULINT := ULINT#4294944000;
	MAX_VALUE_OF_ULINT_WHICH_CAN_BE_HELD_IN_A_DT : ULINT := ULINT#4294967295;
	
	// Limits of REAL used for conversions
	MIN_VALUE_OF_REAL_WHICH_CAN_BE_HELD_IN_A_BYTE : REAL := REAL#0;
	MAX_VALUE_OF_REAL_WHICH_CAN_BE_HELD_IN_A_BYTE : REAL := REAL#255;
	MIN_VALUE_OF_REAL_WHICH_CAN_BE_HELD_IN_A_WORD : REAL := REAL#0;
	MAX_VALUE_OF_REAL_WHICH_CAN_BE_HELD_IN_A_WORD : REAL := REAL#65535;
	MIN_VALUE_OF_REAL_WHICH_CAN_BE_HELD_IN_A_DWORD : REAL := REAL#0;
	MAX_VALUE_OF_REAL_WHICH_CAN_BE_HELD_IN_A_DWORD : REAL := REAL#4.294967E+09;
	MIN_VALUE_OF_REAL_WHICH_CAN_BE_HELD_IN_A_LWORD : REAL := REAL#0;
	MAX_VALUE_OF_REAL_WHICH_CAN_BE_HELD_IN_A_LWORD : REAL := REAL#1.8446743E+19;
	MIN_VALUE_OF_REAL_WHICH_CAN_BE_HELD_IN_A_SINT : REAL := REAL#-128;
	MAX_VALUE_OF_REAL_WHICH_CAN_BE_HELD_IN_A_SINT : REAL := REAL#127;
	MIN_VALUE_OF_REAL_WHICH_CAN_BE_HELD_IN_A_INT : REAL := REAL#-32768;
	MAX_VALUE_OF_REAL_WHICH_CAN_BE_HELD_IN_A_INT : REAL := REAL#32767;
	MIN_VALUE_OF_REAL_WHICH_CAN_BE_HELD_IN_A_DINT : REAL := REAL#-2.14748352E+09;
	MAX_VALUE_OF_REAL_WHICH_CAN_BE_HELD_IN_A_DINT : REAL := REAL#2.14748352E+09;
	MIN_VALUE_OF_REAL_WHICH_CAN_BE_HELD_IN_A_LINT : REAL := REAL#-9.223372E+18;
	MAX_VALUE_OF_REAL_WHICH_CAN_BE_HELD_IN_A_LINT : REAL := REAL#9.223372E+18;
	MIN_VALUE_OF_REAL_WHICH_CAN_BE_HELD_IN_A_USINT : REAL := REAL#0;
	MAX_VALUE_OF_REAL_WHICH_CAN_BE_HELD_IN_A_USINT : REAL := REAL#255;
	MIN_VALUE_OF_REAL_WHICH_CAN_BE_HELD_IN_A_UINT : REAL := REAL#0;
	MAX_VALUE_OF_REAL_WHICH_CAN_BE_HELD_IN_A_UINT : REAL := REAL#65535;
	MIN_VALUE_OF_REAL_WHICH_CAN_BE_HELD_IN_A_UDINT : REAL := REAL#0;
	MAX_VALUE_OF_REAL_WHICH_CAN_BE_HELD_IN_A_UDINT : REAL := REAL#4.294967E+09;
	MIN_VALUE_OF_REAL_WHICH_CAN_BE_HELD_IN_A_ULINT : REAL := REAL#0;
	MAX_VALUE_OF_REAL_WHICH_CAN_BE_HELD_IN_A_ULINT : REAL := REAL#1.8446743E+19;
	MIN_VALUE_OF_REAL_WHICH_CAN_BE_HELD_IN_A_TIME : REAL := REAL#0;
	MAX_VALUE_OF_REAL_WHICH_CAN_BE_HELD_IN_A_TIME : REAL := REAL#4.294967E+09;
	MIN_VALUE_OF_REAL_WHICH_CAN_BE_HELD_IN_A_TOD : REAL := REAL#0;
	MAX_VALUE_OF_REAL_WHICH_CAN_BE_HELD_IN_A_TOD : REAL := REAL#8.639999E+07;
	MIN_VALUE_OF_REAL_WHICH_CAN_BE_HELD_IN_A_DATE : REAL := REAL#0;
	MAX_VALUE_OF_REAL_WHICH_CAN_BE_HELD_IN_A_DATE : REAL := REAL#4.294944E+09;
	MIN_VALUE_OF_REAL_WHICH_CAN_BE_HELD_IN_A_DT : REAL := REAL#0;
	MAX_VALUE_OF_REAL_WHICH_CAN_BE_HELD_IN_A_DT : REAL := REAL#4.294967E+09;
	
	// Limits of LREAL used for conversions
	MIN_VALUE_OF_LREAL_WHICH_CAN_BE_HELD_IN_A_BYTE : LREAL := LREAL#0;
	MAX_VALUE_OF_LREAL_WHICH_CAN_BE_HELD_IN_A_BYTE : LREAL := LREAL#255;
	MIN_VALUE_OF_LREAL_WHICH_CAN_BE_HELD_IN_A_WORD : LREAL := LREAL#0;
	MAX_VALUE_OF_LREAL_WHICH_CAN_BE_HELD_IN_A_WORD : LREAL := LREAL#65535;
	MIN_VALUE_OF_LREAL_WHICH_CAN_BE_HELD_IN_A_DWORD : LREAL := LREAL#0;
	MAX_VALUE_OF_LREAL_WHICH_CAN_BE_HELD_IN_A_DWORD : LREAL := LREAL#4294967295;
	MIN_VALUE_OF_LREAL_WHICH_CAN_BE_HELD_IN_A_LWORD : LREAL := LREAL#0;
	MAX_VALUE_OF_LREAL_WHICH_CAN_BE_HELD_IN_A_LWORD : LREAL := LREAL#1.844674407370955E+19;
	MIN_VALUE_OF_LREAL_WHICH_CAN_BE_HELD_IN_A_SINT : LREAL := LREAL#-128;
	MAX_VALUE_OF_LREAL_WHICH_CAN_BE_HELD_IN_A_SINT : LREAL := LREAL#127;
	MIN_VALUE_OF_LREAL_WHICH_CAN_BE_HELD_IN_A_INT : LREAL := LREAL#-32768;
	MAX_VALUE_OF_LREAL_WHICH_CAN_BE_HELD_IN_A_INT : LREAL := LREAL#32767;
	MIN_VALUE_OF_LREAL_WHICH_CAN_BE_HELD_IN_A_DINT : LREAL := LREAL#-2147483648;
	MAX_VALUE_OF_LREAL_WHICH_CAN_BE_HELD_IN_A_DINT : LREAL := LREAL#2147483647;
	MIN_VALUE_OF_LREAL_WHICH_CAN_BE_HELD_IN_A_LINT : LREAL := LREAL#-9.2233720368547758E+18;
	MAX_VALUE_OF_LREAL_WHICH_CAN_BE_HELD_IN_A_LINT : LREAL := LREAL#9.2233720368547758E+18;
	MIN_VALUE_OF_LREAL_WHICH_CAN_BE_HELD_IN_A_USINT : LREAL := LREAL#0;
	MAX_VALUE_OF_LREAL_WHICH_CAN_BE_HELD_IN_A_USINT : LREAL := LREAL#255;
	MIN_VALUE_OF_LREAL_WHICH_CAN_BE_HELD_IN_A_UINT : LREAL := LREAL#0;
	MAX_VALUE_OF_LREAL_WHICH_CAN_BE_HELD_IN_A_UINT : LREAL := LREAL#65535;
	MIN_VALUE_OF_LREAL_WHICH_CAN_BE_HELD_IN_A_UDINT : LREAL := LREAL#0;
	MAX_VALUE_OF_LREAL_WHICH_CAN_BE_HELD_IN_A_UDINT : LREAL := LREAL#4294967295;
	MIN_VALUE_OF_LREAL_WHICH_CAN_BE_HELD_IN_A_ULINT : LREAL := LREAL#0;
	MAX_VALUE_OF_LREAL_WHICH_CAN_BE_HELD_IN_A_ULINT : LREAL := LREAL#1.844674407370955E+19;
	MIN_VALUE_OF_LREAL_WHICH_CAN_BE_HELD_IN_A_REAL : LREAL := LREAL#-3.402823E+38;
	MAX_VALUE_OF_LREAL_WHICH_CAN_BE_HELD_IN_A_REAL : LREAL := LREAL#3.402823E+38;
	MIN_VALUE_OF_LREAL_WHICH_CAN_BE_HELD_IN_A_TIME : LREAL := LREAL#0;
	MAX_VALUE_OF_LREAL_WHICH_CAN_BE_HELD_IN_A_TIME : LREAL := LREAL#4294967295;
	MIN_VALUE_OF_LREAL_WHICH_CAN_BE_HELD_IN_A_TOD : LREAL := LREAL#0;
	MAX_VALUE_OF_LREAL_WHICH_CAN_BE_HELD_IN_A_TOD : LREAL := LREAL#86399999;
	MIN_VALUE_OF_LREAL_WHICH_CAN_BE_HELD_IN_A_DATE : LREAL := LREAL#0;
	MAX_VALUE_OF_LREAL_WHICH_CAN_BE_HELD_IN_A_DATE : LREAL := LREAL#4294944000;
	MIN_VALUE_OF_LREAL_WHICH_CAN_BE_HELD_IN_A_DT : LREAL := LREAL#0;
	MAX_VALUE_OF_LREAL_WHICH_CAN_BE_HELD_IN_A_DT : LREAL := LREAL#4294967295;
	MAX_VALUE_OF_LREAL_WHICH_CAN_BE_HELD_IN_A_STRING : LREAL := LREAL#9.999999999999E+307; // not sure why this is the number and not LREAL#4.94065645841247E-324.
	MIN_VALUE_OF_LREAL_WHICH_CAN_BE_HELD_IN_A_STRING : LREAL := LREAL#-9.999999999999E+307; // not sure why this is the number and not LREAL#-4.94065645841247E-324.
	
	// Limits of TIME used for conversions
	MAX_VALUE_OF_TIME_WHICH_CAN_BE_HELD_IN_A_BYTE : TIME := T#255MS;
	MAX_VALUE_OF_TIME_WHICH_CAN_BE_HELD_IN_A_WORD : TIME := T#1M5S535MS;
	MAX_VALUE_OF_TIME_WHICH_CAN_BE_HELD_IN_A_SINT : TIME := T#127MS;
	MAX_VALUE_OF_TIME_WHICH_CAN_BE_HELD_IN_A_INT : TIME := T#32S767MS;
	MAX_VALUE_OF_TIME_WHICH_CAN_BE_HELD_IN_A_DINT : TIME := T#24D20H31M23S647MS;
	MAX_VALUE_OF_TIME_WHICH_CAN_BE_HELD_IN_A_USINT : TIME := T#255MS;
	MAX_VALUE_OF_TIME_WHICH_CAN_BE_HELD_IN_A_UINT : TIME := T#1M5S535MS;
	MAX_VALUE_OF_TIME_WHICH_CAN_BE_HELD_IN_A_TOD : TIME := T#23H59M59S999MS;
	
	// Limits of TOD used for conversions
	MAX_VALUE_OF_TOD_WHICH_CAN_BE_HELD_IN_A_BYTE : TOD := TOD#0:0:0.255;
	MAX_VALUE_OF_TOD_WHICH_CAN_BE_HELD_IN_A_WORD : TOD := TOD#0:1:5.535;
	MAX_VALUE_OF_TOD_WHICH_CAN_BE_HELD_IN_A_SINT : TOD := TOD#0:0:0.127;
	MAX_VALUE_OF_TOD_WHICH_CAN_BE_HELD_IN_A_INT : TOD := TOD#0:0:32.767;
	MAX_VALUE_OF_TOD_WHICH_CAN_BE_HELD_IN_A_USINT : TOD := TOD#0:0:0.255;
	MAX_VALUE_OF_TOD_WHICH_CAN_BE_HELD_IN_A_UINT : TOD := TOD#0:1:5.535;
	
	// Limits of DATE used for conversions
	MAX_VALUE_OF_DATE_WHICH_CAN_BE_HELD_IN_A_BYTE : DATE := D#1970-1-1;
	MAX_VALUE_OF_DATE_WHICH_CAN_BE_HELD_IN_A_WORD : DATE := D#1970-1-1;
	MAX_VALUE_OF_DATE_WHICH_CAN_BE_HELD_IN_A_SINT : DATE := D#1970-1-1;
	MAX_VALUE_OF_DATE_WHICH_CAN_BE_HELD_IN_A_INT : DATE := D#1970-1-1;
	MAX_VALUE_OF_DATE_WHICH_CAN_BE_HELD_IN_A_DINT : DATE := D#2038-1-19;
	MAX_VALUE_OF_DATE_WHICH_CAN_BE_HELD_IN_A_USINT : DATE := D#1970-1-1;
	MAX_VALUE_OF_DATE_WHICH_CAN_BE_HELD_IN_A_UINT : DATE := D#1970-1-1;
	MAX_VALUE_OF_DATE_WHICH_CAN_BE_HELD_IN_A_TIME : DATE := D#1970-2-19;
	MAX_VALUE_OF_DATE_WHICH_CAN_BE_HELD_IN_A_TOD : DATE := D#1970-1-1;
	MAX_VALUE_OF_DATE_WHICH_CAN_BE_HELD_IN_A_DT : DATE := D#2106-2-7;
	
	// Limits of DT used for conversions
	MAX_VALUE_OF_DT_WHICH_CAN_BE_HELD_IN_A_BYTE : DT := DT#1970-1-1-0:4:15;
	MAX_VALUE_OF_DT_WHICH_CAN_BE_HELD_IN_A_WORD : DT := DT#1970-1-1-18:12:15;
	MAX_VALUE_OF_DT_WHICH_CAN_BE_HELD_IN_A_SINT : DT := DT#1970-1-1-0:2:7;
	MAX_VALUE_OF_DT_WHICH_CAN_BE_HELD_IN_A_INT : DT := DT#1970-1-1-9:6:7;
	MAX_VALUE_OF_DT_WHICH_CAN_BE_HELD_IN_A_DINT : DT := DT#2038-1-19-3:14:7;
	MAX_VALUE_OF_DT_WHICH_CAN_BE_HELD_IN_A_USINT : DT := DT#1970-1-1-0:4:15;
	MAX_VALUE_OF_DT_WHICH_CAN_BE_HELD_IN_A_UINT : DT := DT#1970-1-1-18:12:15;
	MAX_VALUE_OF_DT_WHICH_CAN_BE_HELD_IN_A_TIME : DT := DT#1970-2-19-17:2:47;
	MAX_VALUE_OF_DT_WHICH_CAN_BE_HELD_IN_A_TOD : DT := DT#1970-1-1-23:59:59;

END_VAR

// ---- mobject-collections/Interfaces/Collections/I_Collection.TcIO
INTERFACE I_Collection EXTENDS I_Enumerable, I_Disposable, I_EventEmitter

METHOD PUBLIC AddItem
VAR_INPUT
	Item : ANY;
END_VAR
END_METHOD

METHOD PUBLIC Clear
END_METHOD

METHOD PUBLIC Contains : BOOL;
VAR_INPUT
	Item : ANY;
END_VAR
END_METHOD

PROPERTY PUBLIC Count : DINT
GET
END_GET
END_PROPERTY

PROPERTY IsEmpty : BOOL
GET
END_GET
END_PROPERTY

METHOD PUBLIC TryCopyTo : BOOL
VAR_INPUT
	Destination : ANY;
END_VAR
END_METHOD

METHOD PUBLIC TryCopyToLocation : BOOL
VAR_INPUT
	DestinationAddress : PVOID;
	DestinationSize : UDINT;
END_VAR
END_METHOD

METHOD PUBLIC TryRemoveItem : BOOL
VAR_INPUT
	Item : ANY;
END_VAR
END_METHOD

END_INTERFACE

// ---- mobject-collections/Interfaces/Collections/I_LinkedList.TcIO
INTERFACE I_LinkedList EXTENDS I_Collection

METHOD PUBLIC AddAfter
VAR_INPUT
	After : I_LinkedListNode;
	Value : ANY;
END_VAR
END_METHOD

METHOD PUBLIC AddBefore
VAR_INPUT
	Before : I_LinkedListNode;
	Value : ANY;
END_VAR
END_METHOD

METHOD PUBLIC AddFirst
VAR_INPUT
	Value : ANY;
END_VAR
END_METHOD

METHOD PUBLIC AddLast
VAR_INPUT
	Value : ANY;
END_VAR
END_METHOD

METHOD PUBLIC Find : I_LinkedListNode
VAR_INPUT
	Value : ANY;
END_VAR
END_METHOD

METHOD PUBLIC FindLast : I_LinkedListNode
VAR_INPUT
	Value : ANY;
END_VAR
END_METHOD

PROPERTY PUBLIC First : I_LinkedListNode
GET
END_GET
END_PROPERTY

PROPERTY PUBLIC Last : I_LinkedListNode
GET
END_GET
END_PROPERTY

METHOD PUBLIC Remove
VAR_INPUT
	Value : ANY;
END_VAR
END_METHOD

METHOD PUBLIC RemoveFirst
END_METHOD

METHOD PUBLIC RemoveLast
END_METHOD

END_INTERFACE

// ---- mobject-collections/Interfaces/Collections/I_Stack.TcIO
INTERFACE I_Stack EXTENDS I_Collection

METHOD PUBLIC Push
VAR_INPUT
	Item : ANY;
END_VAR
END_METHOD

METHOD PUBLIC TryPeek : BOOL;
VAR_INPUT
	Destination : ANY;
END_VAR
END_METHOD

METHOD PUBLIC TryPop : BOOL;
VAR_INPUT
	Destination : ANY;
END_VAR
END_METHOD

END_INTERFACE

// ---- mobject-collections/Interfaces/KeyValueCollections/Nodes/I_DictionaryTreeNode.TcIO
INTERFACE I_DictionaryTreeNode EXTENDS I_CollectionNode

METHOD PUBLIC DeepCopy
VAR_INPUT
	Node : I_DictionaryTreeNode;
END_VAR
END_METHOD

PROPERTY PUBLIC Height : DINT
GET
END_GET
SET
END_SET
END_PROPERTY

PROPERTY PUBLIC Key : T_MAXSTRING
GET
END_GET
END_PROPERTY

PROPERTY PUBLIC Left : I_DictionaryTreeNode
GET
END_GET
SET
END_SET
END_PROPERTY

PROPERTY PUBLIC NodeBufferPointer : Pointer To Byte
GET
END_GET
END_PROPERTY

PROPERTY PUBLIC NodeBufferSize : UDINT
GET
END_GET
END_PROPERTY

METHOD Reinitialize
VAR_INPUT
	Key : T_MAXSTRING;
	Source : ANY;
END_VAR
END_METHOD

PROPERTY PUBLIC Right : I_DictionaryTreeNode
GET
END_GET
SET
END_SET
END_PROPERTY

END_INTERFACE

// ---- mobject-collections/Interfaces/KeyValueCollections/Nodes/I_OrderedDictionaryTreeNode.TcIO
INTERFACE I_OrderedDictionaryTreeNode EXTENDS I_CollectionNode

METHOD PUBLIC DeepCopy
VAR_INPUT
	Node : I_OrderedDictionaryTreeNode;
END_VAR
END_METHOD

PROPERTY PUBLIC Height : DINT
GET
END_GET
SET
END_SET
END_PROPERTY

PROPERTY PUBLIC Key : T_MAXSTRING
GET
END_GET
END_PROPERTY

PROPERTY PUBLIC Left : I_OrderedDictionaryTreeNode
GET
END_GET
SET
END_SET
END_PROPERTY

PROPERTY PUBLIC Next : I_OrderedDictionaryTreeNode
GET
END_GET
SET
END_SET
END_PROPERTY

PROPERTY PUBLIC NodeBufferPointer : Pointer To Byte
GET
END_GET
END_PROPERTY

PROPERTY PUBLIC NodeBufferSize : UDINT
GET
END_GET
END_PROPERTY

PROPERTY PUBLIC Previous : I_OrderedDictionaryTreeNode
GET
END_GET
SET
END_SET
END_PROPERTY

METHOD Reinitialize
VAR_INPUT
	Key : T_MAXSTRING;
	Source : ANY;
END_VAR
END_METHOD

PROPERTY PUBLIC Right : I_OrderedDictionaryTreeNode
GET
END_GET
SET
END_SET
END_PROPERTY

END_INTERFACE

// ---- mobject-commands/AsyncCommand/Interface/I_AsyncCommand.TcIO
INTERFACE I_AsyncCommand extends I_Command

METHOD PUBLIC Abort
VAR_INPUT
END_VAR
END_METHOD

PROPERTY PUBLIC Busy : BOOL
GET
END_GET
END_PROPERTY

METHOD PUBLIC CyclicCall
VAR_INPUT
END_VAR
END_METHOD

PROPERTY PUBLIC Done : BOOL
GET
END_GET
END_PROPERTY

PROPERTY PUBLIC Error : BOOL
GET
END_GET
END_PROPERTY

PROPERTY PUBLIC ErrorId : UDINT
GET
END_GET
END_PROPERTY

END_INTERFACE

// ---- mobject-commands/Command/Interface/I_Command.TcIO
INTERFACE I_Command EXTENDS I_Disposable

METHOD Execute
VAR_INPUT
END_VAR
END_METHOD

END_INTERFACE

// ---- mobject-datatypes/DatatypeOperations/Interface/I_DatatypeOperation.TcIO
INTERFACE I_DatatypeOperation EXTENDS I_Disposable

METHOD Execute
VAR
END_VAR
END_METHOD

END_INTERFACE

// ---- mobject-datatypes/Datatypes/Events/I_AliasDatatypeAddedEvent.TcIO
INTERFACE I_AliasDatatypeAddedEvent EXTENDS I_Event

PROPERTY PUBLIC Target : I_AliasDatatype
GET
END_GET
END_PROPERTY

END_INTERFACE

// ---- mobject-datatypes/Datatypes/Events/I_InterfaceDatatypeAddedEvent.TcIO
INTERFACE I_InterfaceDatatypeAddedEvent EXTENDS I_Event

PROPERTY PUBLIC Target : I_InterfaceDatatype
GET
END_GET
END_PROPERTY

END_INTERFACE

// ---- mobject-datatypes/Datatypes/Events/I_StructuredDatatypeAddedEvent.TcIO
INTERFACE I_StructuredDatatypeAddedEvent EXTENDS I_Event

PROPERTY PUBLIC Target : I_StructuredDatatype
GET
END_GET
END_PROPERTY

END_INTERFACE

// ---- mobject-datatypes/Datatypes/Events/I_ArrayDatatypeAddedEvent.TcIO
INTERFACE I_ArrayDatatypeAddedEvent EXTENDS I_Event

PROPERTY PUBLIC Target : I_ArrayDatatype
GET
END_GET
END_PROPERTY

END_INTERFACE

// ---- mobject-datatypes/Datatypes/Interface/I_Datatypes.TcIO
INTERFACE I_Datatypes EXTENDS I_EventEmitter

METHOD PUBLIC Accept
VAR_INPUT
	Visitor : I_DatatypeVisitor;
END_VAR
END_METHOD

METHOD PUBLIC GetAliasByIdentifier : BOOL
VAR_INPUT
	Identifier : T_MAXSTRING;
	Destination : REFERENCE TO I_AliasDatatype;
END_VAR
END_METHOD

METHOD PUBLIC GetPrimitiveByTypeName : BOOL
VAR_INPUT
	TypeName : T_MAXSTRING;
	Destination : REFERENCE TO I_AliasDatatype;
END_VAR
END_METHOD

METHOD PUBLIC GetStructureByIdentifier : BOOL
VAR_INPUT
	Identifier : T_MAXSTRING;
	Destination : REFERENCE TO I_StructuredDatatype;
END_VAR
END_METHOD

METHOD RegisterDatatype
VAR_INPUT
	Datatype : I_Datatype;
END_VAR
END_METHOD

METHOD PUBLIC SerializeTypeWith
VAR_INPUT
	Serializer : I_Serializer;
END_VAR
END_METHOD

END_INTERFACE

// ---- mobject-datatypes/_Internal/Datatype/Interface/I_AliasDatatype.TcIO
INTERFACE I_AliasDatatype EXTENDS I_UserDefinedDatatype

PROPERTY PUBLIC BaseDatatype : I_Datatype
GET
END_GET
END_PROPERTY

PROPERTY PUBLIC RootDatatype : I_Datatype
GET
END_GET
END_PROPERTY

END_INTERFACE

// ---- mobject-datatypes/_Internal/Datatype/Interface/I_ArrayDatatype_2D.TcIO
INTERFACE I_ArrayDatatype_2D EXTENDS I_ArrayDatatype

METHOD PUBLIC TryGetElementAsDatatypeByIndex : BOOL
VAR_INPUT
	Index1 : DINT;
	Index2 : DINT;
	Destination : REFERENCE TO I_Datatype;
END_VAR
END_METHOD

END_INTERFACE

// ---- mobject-datatypes/_Internal/Datatype/Interface/I_BitDatatype.TcIO
INTERFACE I_BitDatatype EXTENDS I_Datatype

PROPERTY PUBLIC BitOffset : DWORD
GET
END_GET
END_PROPERTY

PROPERTY PUBLIC ByteOffset : PVOID
GET
END_GET
END_PROPERTY

PROPERTY PUBLIC Parent : I_StructuredDatatype
GET
END_GET
END_PROPERTY

PROPERTY PUBLIC Value : BOOL
GET
END_GET
SET
END_SET
END_PROPERTY

END_INTERFACE

// ---- mobject-datatypes/_Internal/Datatype/Interface/I_Datatype.TcIO
INTERFACE I_Datatype extends I_Serializable, I_Deserializable, I_Disposable

METHOD PUBLIC Accept
VAR_INPUT
	Visitor : I_DatatypeVisitor;
END_VAR
END_METHOD

PROPERTY PUBLIC Address : PVOID
GET
END_GET
END_PROPERTY

METHOD PUBLIC ClearReference
VAR_INPUT
END_VAR
END_METHOD

METHOD Clone : I_Datatype
END_METHOD

METHOD PUBLIC IsEquivalentTo : BOOL
VAR_INPUT
	Datatype : I_Datatype;
END_VAR
END_METHOD

PROPERTY PUBLIC IsUserDefined : BOOL
GET
END_GET
END_PROPERTY

PROPERTY PUBLIC Root : I_Datatype
GET
END_GET
END_PROPERTY

METHOD PUBLIC SerializeTypeWith
VAR_INPUT
	Serializer : I_Serializer;
END_VAR
END_METHOD

PROPERTY PUBLIC Size : UDINT
GET
END_GET
END_PROPERTY

METHOD PUBLIC TryCopyFrom : BOOL
VAR_INPUT
	Source : I_Datatype;
END_VAR
END_METHOD

METHOD PUBLIC ABSTRACT TryDeserializeFrom : BOOL
VAR_INPUT
	Deserializer : I_Deserializer;
	Feedback : I_DeserializerFeedback;
END_VAR
END_METHOD

METHOD TryMakeReferenceTo : BOOL
VAR_INPUT
	Target : I_Datatype;
END_VAR
END_METHOD

METHOD PUBLIC TryResolveAsAliasDatatype : BOOL
VAR_INPUT
	Destination : REFERENCE TO I_AliasDatatype;
END_VAR
END_METHOD

METHOD PUBLIC TryResolveAsArrayDatatype : BOOL
VAR_INPUT
	Destination : REFERENCE TO I_ArrayDatatype;
END_VAR
END_METHOD

METHOD PUBLIC TryResolveAsBitDatatype : BOOL
VAR_INPUT
	Destination : REFERENCE TO I_BitDatatype;
END_VAR
END_METHOD

METHOD PUBLIC TryResolveAsEnumDatatype : BOOL
VAR_INPUT
	Destination : REFERENCE TO I_EnumDatatype;
END_VAR
END_METHOD

METHOD PUBLIC TryResolveAsInterfaceDatatype : BOOL
VAR_INPUT
	Destination : REFERENCE TO I_InterfaceDatatype;
END_VAR
END_METHOD

METHOD PUBLIC TryResolveAsStructuredDatatype : BOOL
VAR_INPUT
	Destination : REFERENCE TO I_StructuredDatatype;
END_VAR
END_METHOD

METHOD PUBLIC TryResolveAsUserDefinedDatatype : BOOL
VAR_INPUT
	Destination : REFERENCE TO I_UserDefinedDatatype;
END_VAR
END_METHOD

PROPERTY PUBLIC TypeName : T_MAXSTRING
GET
END_GET
END_PROPERTY

END_INTERFACE

// ---- mobject-datatypes/_Internal/Datatype/Interface/I_NumericDatatype.TcIO
INTERFACE I_NumericDatatype EXTENDS I_Datatype

PROPERTY PUBLIC ABSTRACT IsFloat : BOOL
GET
END_GET
END_PROPERTY

PROPERTY PUBLIC IsSigned : BOOL
GET
END_GET
END_PROPERTY

END_INTERFACE

// ---- mobject-datatypes/_Internal/Datatype/Interface/I_ArrayDatatype.TcIO
INTERFACE I_ArrayDatatype EXTENDS I_UserDefinedDatatype

METHOD PUBLIC ABSTRACT GetElementAsDatatypeByIndex : I_Datatype
VAR_INPUT
	Index : DINT;
END_VAR
END_METHOD

PROPERTY PUBLIC ABSTRACT LowerBound : DINT
GET
END_GET
END_PROPERTY

PROPERTY PUBLIC ABSTRACT UpperBound : DINT
GET
END_GET
END_PROPERTY

END_INTERFACE

// ---- mobject-datatypes/_Internal/StructureMembers/Interface/I_StructureMembers.TcIO
INTERFACE I_StructureMembers

METHOD PUBLIC Accept
VAR_INPUT
	Visitor : I_DatatypeVisitor;
END_VAR
END_METHOD

METHOD PUBLIC GetMemberEnumerator : I_KeyValueForwardEnumerator
VAR_INPUT
END_VAR
END_METHOD

METHOD PUBLIC TryGetMemberByName : BOOL
VAR_INPUT
	Name : T_MAXSTRING;
	Destination : REFERENCE TO I_Datatype;
END_VAR
END_METHOD

END_INTERFACE

// ---- mobject-deserialization/GarbageCollector/I_DeserializerGarbageCollector.TcIO
INTERFACE I_DeserializerGarbageCollector EXTENDS __SYSTEM.IQueryInterface

METHOD PUBLIC Deregister
VAR_INPUT
	Deserializer : I_Deserializer;
END_VAR
END_METHOD

METHOD PUBLIC Register
VAR_INPUT
	Deserializer : I_Deserializer;
END_VAR
END_METHOD

END_INTERFACE

// ---- mobject-deserialization/Interfaces/I_Deserializable.TcIO
INTERFACE I_Deserializable EXTENDS __SYSTEM.IQueryInterface

METHOD TryDeserializeFrom : BOOL
VAR_INPUT
	Deserializer : I_Deserializer;
	Feedback : I_DeserializerFeedback;
END_VAR
END_METHOD

END_INTERFACE

// ---- mobject-deserialization/Interfaces/I_Deserializer.TcIO
INTERFACE I_Deserializer EXTENDS I_Disposable

METHOD PUBLIC Clone : I_Deserializer
END_METHOD

METHOD GetArray : I_Deserializer
VAR_INPUT
END_VAR
END_METHOD

METHOD GetArrayEnumerator : I_DeserializerArrayForwardEnumerator
VAR_INPUT
END_VAR
END_METHOD

METHOD GetElementByIndex : I_Deserializer
VAR_INPUT
	Index : UDINT;
END_VAR
END_METHOD

METHOD GetKeyArray : I_Deserializer
VAR_INPUT
	Key : T_MAXSTRING;
END_VAR
END_METHOD

METHOD GetKeyObject : I_Deserializer
VAR_INPUT
	Key : T_MAXSTRING;
END_VAR
END_METHOD

METHOD GetObject : I_Deserializer
VAR_INPUT
END_VAR
END_METHOD

METHOD GetObjectEnumerator : I_DeserializerObjectForwardEnumerator
VAR_INPUT
END_VAR
END_METHOD

METHOD TryDeserializeKeyToObject : BOOL
VAR_INPUT
	Key : T_MAXSTRING;
	Object : I_Deserializable;
	Feedback : I_DeserializerFeedback;
END_VAR
END_METHOD

METHOD TryDeserializeToObject : BOOL
VAR_INPUT
	Object : I_Deserializable;
	Feedback : I_DeserializerFeedback;
END_VAR
END_METHOD

METHOD TryGetBase64 : BOOL
VAR_INPUT
	pBytes : POINTER TO BYTE;
	nBytes : DINT;
	Feedback : I_DeserializerFeedback;
END_VAR
END_METHOD

METHOD TryGetBool : BOOL
VAR_INPUT
	Destination : REFERENCE TO BOOL;
	Feedback : I_DeserializerFeedback;
END_VAR
END_METHOD

METHOD TryGetByte : BOOL
VAR_INPUT
	Destination : REFERENCE TO BYTE;
	Feedback : I_DeserializerFeedback;
END_VAR
END_METHOD

METHOD TryGetDateTime : BOOL
VAR_INPUT
	Destination : REFERENCE TO DATE_AND_TIME;
	Feedback : I_DeserializerFeedback;
END_VAR
END_METHOD

METHOD TryGetDcTime : BOOL
VAR_INPUT
	Destination : REFERENCE TO DCTIME;
	Feedback : I_DeserializerFeedback;
END_VAR
END_METHOD

METHOD TryGetDint : BOOL
VAR_INPUT
	Destination : REFERENCE TO DINT;
	Feedback : I_DeserializerFeedback;
END_VAR
END_METHOD

METHOD TryGetDword : BOOL
VAR_INPUT
	Destination : REFERENCE TO DWORD;
	Feedback : I_DeserializerFeedback;
END_VAR
END_METHOD

METHOD TryGetFileTime : BOOL
VAR_INPUT
	Destination : REFERENCE TO FILETIME;
	Feedback : I_DeserializerFeedback;
END_VAR
END_METHOD

METHOD TryGetHexAsBytes : BOOL
VAR_INPUT
	pBytes : POINTER TO BYTE;
	nBytes : DINT;
	Feedback : I_DeserializerFeedback;
END_VAR
END_METHOD

METHOD TryGetInt : BOOL
VAR_INPUT
	Destination : REFERENCE TO INT;
	Feedback : I_DeserializerFeedback;
END_VAR
END_METHOD

METHOD TryGetKeyBase64 : BOOL
VAR_INPUT
	Key : T_MAXSTRING;
	pBytes : POINTER TO BYTE;
	nBytes : DINT;
	Feedback : I_DeserializerFeedback;
END_VAR
END_METHOD

METHOD TryGetKeyBool : BOOL
VAR_INPUT
	Key : T_MAXSTRING;
	Destination : REFERENCE TO BOOL;
	Feedback : I_DeserializerFeedback;
END_VAR
END_METHOD

METHOD TryGetKeyByte : BOOL
VAR_INPUT
	Key : T_MAXSTRING;
	Destination : REFERENCE TO BYTE;
	Feedback : I_DeserializerFeedback;
END_VAR
END_METHOD

METHOD TryGetKeyDateTime : BOOL
VAR_INPUT
	Key : T_MAXSTRING;
	Destination : REFERENCE TO DATE_AND_TIME;
	Feedback : I_DeserializerFeedback;
END_VAR
END_METHOD

METHOD TryGetKeyDcTime : BOOL
VAR_INPUT
	Key : T_MAXSTRING;
	Destination : REFERENCE TO DCTIME;
	Feedback : I_DeserializerFeedback;
END_VAR
END_METHOD

METHOD TryGetKeyDint : BOOL
VAR_INPUT
	Key : T_MAXSTRING;
	Destination : REFERENCE TO DINT;
	Feedback : I_DeserializerFeedback;
END_VAR
END_METHOD

METHOD TryGetKeyDword : BOOL
VAR_INPUT
	Key : T_MAXSTRING;
	Destination : REFERENCE TO DWORD;
	Feedback : I_DeserializerFeedback;
END_VAR
END_METHOD

METHOD TryGetKeyFileTime : BOOL
VAR_INPUT
	Key : T_MAXSTRING;
	Destination : REFERENCE TO FILETIME;
	Feedback : I_DeserializerFeedback;
END_VAR
END_METHOD

METHOD TryGetKeyHexAsBytes : BOOL
VAR_INPUT
	Key : T_MAXSTRING;
	pBytes : POINTER TO BYTE;
	nBytes : DINT;
	Feedback : I_DeserializerFeedback;
END_VAR
END_METHOD

METHOD TryGetKeyInt : BOOL
VAR_INPUT
	Key : T_MAXSTRING;
	Destination : REFERENCE TO INT;
	Feedback : I_DeserializerFeedback;
END_VAR
END_METHOD

METHOD TryGetKeyLint : BOOL
VAR_INPUT
	Key : T_MAXSTRING;
	Destination : REFERENCE TO LINT;
	Feedback : I_DeserializerFeedback;
END_VAR
END_METHOD

METHOD TryGetKeyLreal : BOOL
VAR_INPUT
	Key : T_MAXSTRING;
	Destination : REFERENCE TO LREAL;
	Feedback : I_DeserializerFeedback;
END_VAR
END_METHOD

METHOD TryGetKeyLtime : BOOL
VAR_INPUT
	Key : T_MAXSTRING;
	Destination : REFERENCE TO LTIME;
	Feedback : I_DeserializerFeedback;
END_VAR
END_METHOD

METHOD TryGetKeyLword : BOOL
VAR_INPUT
	Key : T_MAXSTRING;
	Destination : REFERENCE TO LWORD;
	Feedback : I_DeserializerFeedback;
END_VAR
END_METHOD

METHOD TryGetKeyReal : BOOL
VAR_INPUT
	Key : T_MAXSTRING;
	Destination : REFERENCE TO REAL;
	Feedback : I_DeserializerFeedback;
END_VAR
END_METHOD

METHOD TryGetKeySint : BOOL
VAR_INPUT
	Key : T_MAXSTRING;
	Destination : REFERENCE TO SINT;
	Feedback : I_DeserializerFeedback;
END_VAR
END_METHOD

METHOD TryGetKeyString : BOOL
VAR_INPUT
	Key : T_MAXSTRING;
	Destination : REFERENCE TO STRING;
	Feedback : I_DeserializerFeedback;
END_VAR
END_METHOD

METHOD TryGetKeyTime : BOOL
VAR_INPUT
	Key : T_MAXSTRING;
	Destination : REFERENCE TO TIME;
	Feedback : I_DeserializerFeedback;
END_VAR
END_METHOD

METHOD TryGetKeyTod : BOOL
VAR_INPUT
	Key : T_MAXSTRING;
	Destination : REFERENCE TO TOD;
	Feedback : I_DeserializerFeedback;
END_VAR
END_METHOD

METHOD TryGetKeyUdint : BOOL
VAR_INPUT
	Key : T_MAXSTRING;
	Destination : REFERENCE TO UDINT;
	Feedback : I_DeserializerFeedback;
END_VAR
END_METHOD

METHOD TryGetKeyUint : BOOL
VAR_INPUT
	Key : T_MAXSTRING;
	Destination : REFERENCE TO UINT;
	Feedback : I_DeserializerFeedback;
END_VAR
END_METHOD

METHOD TryGetKeyUlint : BOOL
VAR_INPUT
	Key : T_MAXSTRING;
	Destination : REFERENCE TO ULINT;
	Feedback : I_DeserializerFeedback;
END_VAR
END_METHOD

METHOD TryGetKeyUsint : BOOL
VAR_INPUT
	Key : T_MAXSTRING;
	Destination : REFERENCE TO USINT;
	Feedback : I_DeserializerFeedback;
END_VAR
END_METHOD

METHOD TryGetKeyWord : BOOL
VAR_INPUT
	Key : T_MAXSTRING;
	Destination : REFERENCE TO WORD;
	Feedback : I_DeserializerFeedback;
END_VAR
END_METHOD

METHOD TryGetLint : BOOL
VAR_INPUT
	Destination : REFERENCE TO LINT;
	Feedback : I_DeserializerFeedback;
END_VAR
END_METHOD

METHOD TryGetLreal : BOOL
VAR_INPUT
	Destination : REFERENCE TO LREAL;
	Feedback : I_DeserializerFeedback;
END_VAR
END_METHOD

METHOD TryGetLtime : BOOL
VAR_INPUT
	Destination : REFERENCE TO LTIME;
	Feedback : I_DeserializerFeedback;
END_VAR
END_METHOD

METHOD TryGetLword : BOOL
VAR_INPUT
	Destination : REFERENCE TO LWORD;
	Feedback : I_DeserializerFeedback;
END_VAR
END_METHOD

METHOD TryGetReal : BOOL
VAR_INPUT
	Destination : REFERENCE TO REAL;
	Feedback : I_DeserializerFeedback;
END_VAR
END_METHOD

METHOD TryGetSint : BOOL
VAR_INPUT
	Destination : REFERENCE TO SINT;
	Feedback : I_DeserializerFeedback;
END_VAR
END_METHOD

METHOD TryGetString : BOOL
VAR_INPUT
	Destination : REFERENCE TO STRING;
	Feedback : I_DeserializerFeedback;
END_VAR
END_METHOD

METHOD TryGetTime : BOOL
VAR_INPUT
	Destination : REFERENCE TO TIME;
	Feedback : I_DeserializerFeedback;
END_VAR
END_METHOD

METHOD TryGetTod : BOOL
VAR_INPUT
	Destination : REFERENCE TO TOD;
	Feedback : I_DeserializerFeedback;
END_VAR
END_METHOD

METHOD TryGetUdint : BOOL
VAR_INPUT
	Destination : REFERENCE TO UDINT;
	Feedback : I_DeserializerFeedback;
END_VAR
END_METHOD

METHOD TryGetUint : BOOL
VAR_INPUT
	Destination : REFERENCE TO UINT;
	Feedback : I_DeserializerFeedback;
END_VAR
END_METHOD

METHOD TryGetUlint : BOOL
VAR_INPUT
	Destination : REFERENCE TO ULINT;
	Feedback : I_DeserializerFeedback;
END_VAR
END_METHOD

METHOD TryGetUsint : BOOL
VAR_INPUT
	Destination : REFERENCE TO USINT;
	Feedback : I_DeserializerFeedback;
END_VAR
END_METHOD

METHOD TryGetWord : BOOL
VAR_INPUT
	Destination : REFERENCE TO WORD;
	Feedback : I_DeserializerFeedback;
END_VAR
END_METHOD

END_INTERFACE

// ---- mobject-events/Interfaces/I_EventEmitter.TcIO
INTERFACE I_EventEmitter EXTENDS __SYSTEM.IQueryInterface

METHOD PUBLIC OffEvent
VAR_INPUT
	EventName : T_MaxString;
	EventHandler : I_EventHandler;
END_VAR
END_METHOD

METHOD PUBLIC OnceEvent
VAR_INPUT
	EventName : T_MaxString;
	EventHandler : I_EventHandler;
END_VAR
END_METHOD

METHOD PUBLIC OnEvent
VAR_INPUT
	EventName : T_MaxString;
	EventHandler : I_EventHandler;
END_VAR
END_METHOD

END_INTERFACE

// ---- mobject-events/Interfaces/I_EventHandler.TcIO
INTERFACE I_EventHandler EXTENDS __SYSTEM.IQueryInterface

METHOD PUBLIC HandleEvent
VAR_INPUT
	Event : I_Event;
END_VAR
END_METHOD

END_INTERFACE

// ---- mobject-events/Interfaces/I_EventTarget.TcIO
INTERFACE I_EventTarget EXTENDS __SYSTEM.IQueryInterface

METHOD PUBLIC Emit
VAR_INPUT
	EventName : T_MaxString;
	Event : I_Event;
END_VAR
END_METHOD

END_INTERFACE

// ---- mobject-enumerable/Interfaces/Enumerators/I_KeyValueForwardEnumerator.TcIO
INTERFACE I_KeyValueForwardEnumerator EXTENDS I_ForwardEnumerator

PROPERTY Key : T_MAXSTRING
GET
END_GET
END_PROPERTY

END_INTERFACE

// ---- mobject-json/JsonDeserializer/Events/I_JsonDeserializerChangedEvent.TcIO
INTERFACE I_JsonDeserializerChangedEvent EXTENDS I_Event

PROPERTY PUBLIC Target : I_JsonDeserializer
GET
END_GET
END_PROPERTY

END_INTERFACE

// ---- mobject-json/_Internal/JsonPathVisitor/I_JsonPathVisitor.TcIO
INTERFACE I_JsonPathVisitor EXTENDS __System.IQueryInterface

METHOD ArrayIndexFound
VAR_INPUT
	Index : UDINT;
END_VAR
END_METHOD

METHOD EndOfParse
VAR_INPUT
END_VAR
END_METHOD

METHOD InvalidSyntaxFound
VAR_INPUT
	Character : BYTE;
	Position : UDINT;
END_VAR
END_METHOD

METHOD PropertyFound
VAR_INPUT
	Name : T_MAXSTRING;
END_VAR
END_METHOD

METHOD StartOfParse
VAR_INPUT
END_VAR
END_METHOD

END_INTERFACE

// ---- mobject-datatypes/Datatypes/Base/Datatypes.TcPOU
{attribute 'linkalways'} 
{attribute 'no_explicit_call' := 'This FB is a CLASS and must be accessed using methods or properties'}
{attribute 'enable_dynamic_creation'}
FUNCTION_BLOCK Datatypes IMPLEMENTS I_Datatypes
VAR
	eventEmitter : EventEmitter;
	primitives : Dictionary;
	structures : Dictionary;
	arrays : Dictionary;
	alias : Dictionary;
	enums : Dictionary;
	interfaces : Dictionary;
END_VAR

METHOD PUBLIC Accept
VAR_INPUT
	Visitor : I_DatatypeVisitor;
END_VAR
AcceptPrimative(Visitor);
AcceptStructures(Visitor);
AcceptArrays(Visitor);
AcceptAlias(Visitor);
AcceptEnum(Visitor);
AcceptInterface(Visitor);
END_METHOD

METHOD PRIVATE AcceptAlias
VAR_INPUT
	Visitor : I_DatatypeVisitor;
END_VAR
VAR
	enumerator : I_ForwardEnumerator;
	datatype : I_AliasDatatype;
END_VAR
enumerator := alias.GetEnumerator();

WHILE enumerator.MoveNext() DO
	IF enumerator.TryGet(datatype) THEN
		datatype.Accept(Visitor);
	END_IF
END_WHILE

enumerator.Dispose();
END_METHOD

METHOD PRIVATE AcceptArrays
VAR_INPUT
	Visitor : I_DatatypeVisitor;
END_VAR
VAR
	enumerator : I_ForwardEnumerator;
	datatype : I_ArrayDatatype;
END_VAR
enumerator := arrays.GetEnumerator();

WHILE enumerator.MoveNext() DO	
	IF enumerator.TryGet(datatype) THEN
		datatype.Accept(Visitor);
	END_IF
END_WHILE

enumerator.Dispose();
END_METHOD

METHOD PRIVATE AcceptEnum
VAR_INPUT
	Visitor : I_DatatypeVisitor;
END_VAR
VAR
	enumerator : I_ForwardEnumerator;
	datatype : I_EnumDatatype;
END_VAR
enumerator := enums.GetEnumerator();

WHILE enumerator.MoveNext() DO
	IF enumerator.TryGet(datatype) THEN
		datatype.Accept(Visitor);
	END_IF
END_WHILE

enumerator.Dispose();
END_METHOD

METHOD PRIVATE AcceptInterface
VAR_INPUT
	Visitor : I_DatatypeVisitor;
END_VAR
VAR
	enumerator : I_ForwardEnumerator;
	datatype : I_InterfaceDatatype;
END_VAR
enumerator := structures.GetEnumerator();

WHILE enumerator.MoveNext() DO	
	IF enumerator.TryGet(datatype) THEN
		datatype.Accept(Visitor);
	END_IF
END_WHILE

enumerator.Dispose();
END_METHOD

METHOD PRIVATE AcceptPrimative
VAR_INPUT
	Visitor : I_DatatypeVisitor;
END_VAR
VAR
	enumerator : I_ForwardEnumerator;
	datatype : I_Datatype;
END_VAR
enumerator := primitives.GetEnumerator();

WHILE enumerator.MoveNext() DO
	IF enumerator.TryGet(datatype) THEN
		datatype.Accept(Visitor);
	END_IF
END_WHILE

enumerator.Dispose();
END_METHOD

METHOD PRIVATE AcceptStructures
VAR_INPUT
	Visitor : I_DatatypeVisitor;
END_VAR
VAR
	enumerator : I_ForwardEnumerator;
	datatype : I_StructuredDatatype;
END_VAR
enumerator := structures.GetEnumerator();

WHILE enumerator.MoveNext() DO	
	IF enumerator.TryGet(datatype) THEN
		datatype.Accept(Visitor);
	END_IF
END_WHILE

enumerator.Dispose();
END_METHOD

METHOD PROTECTED EmitOnAliasDatatypeAddedEvent
VAR_INPUT
	Datatype : I_AliasDatatype;
END_VAR
VAR
	datatypeAddedEvent : AliasDatatypeAddedEvent(Target := Datatype);
END_VAR
eventEmitter.Emit('OnDatatypeAdded', datatypeAddedEvent);
END_METHOD

METHOD PROTECTED EmitOnArrayDatatypeAddedEvent
VAR_INPUT
	Datatype : I_ArrayDatatype;
END_VAR
VAR
	datatypeAddedEvent : ArrayDatatypeAddedEvent(Target := Datatype);
END_VAR
eventEmitter.Emit('OnDatatypeAdded', datatypeAddedEvent);
END_METHOD

METHOD PROTECTED EmitOnDatatypeAddedEvent
VAR_INPUT
	Datatype : I_Datatype;
END_VAR
VAR
	datatypeAddedEvent : DatatypeAddedEvent(Target := Datatype);
END_VAR
eventEmitter.Emit('OnDatatypeAdded', datatypeAddedEvent);
END_METHOD

METHOD PROTECTED EmitOnEnumDatatypeAddedEvent
VAR_INPUT
	Datatype : I_EnumDatatype;
END_VAR
VAR
	datatypeAddedEvent : EnumDatatypeAddedEvent(Target := Datatype);
END_VAR
eventEmitter.Emit('OnDatatypeAdded', datatypeAddedEvent);
END_METHOD

METHOD PROTECTED EmitOnInterfaceDatatypeAddedEvent
VAR_INPUT
	Datatype : I_InterfaceDatatype;
END_VAR
VAR
	datatypeAddedEvent : InterfaceDatatypeAddedEvent(Target := Datatype);
END_VAR
eventEmitter.Emit('OnDatatypeAdded', datatypeAddedEvent);
END_METHOD

METHOD PROTECTED EmitOnStructuredDatatypeAddedEvent
VAR_INPUT
	Datatype : I_StructuredDatatype;
END_VAR
VAR
	datatypeAddedEvent : StructuredDatatypeAddedEvent(Target := Datatype);
END_VAR
eventEmitter.Emit('OnDatatypeAdded', datatypeAddedEvent);
END_METHOD

METHOD PUBLIC OffEvent
VAR_INPUT
	EventName : T_MaxString;
	EventHandler : I_EventHandler;
END_VAR
eventEmitter.OffEvent(EventName, EventHandler);
END_METHOD

METHOD PUBLIC OnceEvent
VAR_INPUT
	EventName : T_MaxString;
	EventHandler : I_EventHandler;
END_VAR
eventEmitter.OnceEvent(EventName, EventHandler);
END_METHOD

METHOD PUBLIC OnEvent
VAR_INPUT
	EventName : T_MaxString;
	EventHandler : I_EventHandler;
END_VAR
eventEmitter.OnEvent(EventName, EventHandler);
END_METHOD

METHOD RegisterDatatype
VAR_INPUT
	Datatype : I_Datatype;
END_VAR
VAR
	datatypeAsStructure : I_StructuredDatatype;
	datatypeAsArray : I_ArrayDatatype;
	datatypeAsAlias : I_AliasDatatype;
	datatypeAsEnum : I_EnumDatatype;
	datatypeAsInterface : I_InterfaceDatatype;
END_VAR
IF Datatype.TryResolveAsStructuredDatatype(datatypeAsStructure) THEN
	structures.AddOrUpdate(datatypeAsStructure.Identifier, datatypeAsStructure);
	emitOnStructuredDatatypeAddedEvent(datatypeAsStructure);
	RETURN;
END_IF

IF Datatype.TryResolveAsArrayDatatype(datatypeAsArray) THEN
	arrays.AddOrUpdate(datatypeAsArray.Identifier, datatypeAsArray);
	emitOnArrayDatatypeAddedEvent(datatypeAsArray);
	RETURN;
END_IF

IF Datatype.TryResolveAsAliasDatatype(datatypeAsAlias) THEN
	alias.AddOrUpdate(datatypeAsAlias.Identifier, datatypeAsAlias);
	emitOnAliasDatatypeAddedEvent(datatypeAsAlias);
	RETURN;
END_IF

IF Datatype.TryResolveAsEnumDatatype(datatypeAsEnum) THEN
	enums.AddOrUpdate(datatypeAsEnum.Identifier, datatypeAsEnum);
	emitOnEnumDatatypeAddedEvent(datatypeAsEnum);
	RETURN;
END_IF

IF Datatype.TryResolveAsInterfaceDatatype(datatypeAsInterface) THEN
	interfaces.AddOrUpdate(datatypeAsInterface.Identifier, datatypeAsInterface);
	emitOnInterfaceDatatypeAddedEvent(datatypeAsInterface);
	RETURN;
END_IF

primitives.AddOrUpdate(Datatype.TypeName, Datatype);
emitOnDatatypeAddedEvent(Datatype);
END_METHOD

METHOD PRIVATE SerializeAliasTypeWith
VAR_INPUT
	Serializer : I_Serializer;
END_VAR
VAR
	enumerator : I_ForwardEnumerator;
	datatype : I_AliasDatatype;
END_VAR
enumerator := alias.GetEnumerator();

WHILE enumerator.MoveNext() DO
	IF enumerator.TryGet(datatype) THEN
		datatype.SerializeTypeWith(Serializer);
	END_IF
END_WHILE

enumerator.Dispose();
END_METHOD

METHOD PRIVATE SerializeArrayTypeWith
VAR_INPUT
	Serializer : I_Serializer;
END_VAR
VAR
	enumerator : I_ForwardEnumerator;
	datatype : I_ArrayDatatype;
END_VAR
enumerator := arrays.GetEnumerator();

WHILE enumerator.MoveNext() DO
	IF enumerator.TryGet(datatype) THEN
		datatype.SerializeTypeWith(Serializer);
	END_IF
END_WHILE

enumerator.Dispose();
END_METHOD

METHOD PRIVATE SerializeEnumsTypeWith
VAR_INPUT
	Serializer : I_Serializer;
END_VAR
VAR
	enumerator : I_ForwardEnumerator;
	datatype : I_EnumDatatype;
END_VAR
enumerator := enums.GetEnumerator();

WHILE enumerator.MoveNext() DO
	IF enumerator.TryGet(datatype) THEN
		datatype.SerializeTypeWith(Serializer);
	END_IF
END_WHILE

enumerator.Dispose();
END_METHOD

METHOD PRIVATE SerializeInterfaceTypeWith
VAR_INPUT
	Serializer : I_Serializer;
END_VAR
VAR
	enumerator : I_ForwardEnumerator;
	datatype : I_InterfaceDatatype;
END_VAR
enumerator := interfaces.GetEnumerator();

WHILE enumerator.MoveNext() DO
	IF enumerator.TryGet(datatype) THEN
		datatype.SerializeTypeWith(Serializer);
	END_IF
END_WHILE

enumerator.Dispose();
END_METHOD

METHOD PRIVATE SerializePrimitiveTypeWith
VAR_INPUT
	Serializer : I_Serializer;
END_VAR
VAR
	enumerator : I_ForwardEnumerator;
	datatype : I_Datatype;
END_VAR
enumerator := primitives.GetEnumerator();

WHILE enumerator.MoveNext() DO
	IF enumerator.TryGet(datatype) THEN
		datatype.SerializeTypeWith(Serializer);
	END_IF
END_WHILE

enumerator.Dispose();
END_METHOD

METHOD PRIVATE SerializeStructuresTypeWith
VAR_INPUT
	Serializer : I_Serializer;
END_VAR
VAR
	enumerator : I_ForwardEnumerator;
	datatype : I_StructuredDatatype;
END_VAR
enumerator := structures.GetEnumerator();

WHILE enumerator.MoveNext() DO
	IF enumerator.TryGet(datatype) THEN
		datatype.SerializeTypeWith(Serializer);
	END_IF
END_WHILE

enumerator.Dispose();
END_METHOD

METHOD PUBLIC SerializeTypeWith
VAR_INPUT
	Serializer : I_Serializer;
END_VAR
Serializer.StartObject();
Serializer.AddKey('datatypes');
Serializer.StartArray();
SerializePrimitiveTypeWith(Serializer);
SerializeStructuresTypeWith(Serializer);
SerializeArrayTypeWith(Serializer);
SerializeAliasTypeWith(Serializer);
SerializeEnumsTypeWith(Serializer);
SerializeInterfaceTypeWith(Serializer);
Serializer.EndArray();
Serializer.EndObject();
END_METHOD

METHOD PUBLIC TryGetAliasByIdentifier : BOOL
VAR_INPUT
	Identifier : T_MAXSTRING;
	Destination : REFERENCE TO I_AliasDatatype;
END_VAR
TryGetAliasByIdentifier := alias.TryGetValue(Identifier, Destination);
END_METHOD

METHOD PUBLIC TryGetArrayByIdentifier : BOOL
VAR_INPUT
	Identifier : T_MAXSTRING;
	Destination : REFERENCE TO I_ArrayDatatype;
END_VAR
TryGetArrayByIdentifier := arrays.TryGetValue(Identifier, Destination);
END_METHOD

METHOD PUBLIC TryGetEnumByIdentifier : BOOL
VAR_INPUT
	Identifier : T_MAXSTRING;
	Destination : REFERENCE TO I_EnumDatatype;
END_VAR
TryGetEnumByIdentifier := enums.TryGetValue(Identifier, Destination);
END_METHOD

METHOD PUBLIC TryGetInterfaceByIdentifier : BOOL
VAR_INPUT
	Identifier : T_MAXSTRING;
	Destination : REFERENCE TO I_InterfaceDatatype;
END_VAR
TryGetInterfaceByIdentifier := interfaces.TryGetValue(Identifier, Destination);
END_METHOD

METHOD PUBLIC TryGetPrimitiveByTypeName : BOOL
VAR_INPUT
	TypeName : T_MAXSTRING;
	Destination : REFERENCE TO I_AliasDatatype;
END_VAR
TryGetPrimitiveByTypeName := primitives.TryGetValue(TypeName, Destination);
END_METHOD

METHOD PUBLIC TryGetStructureByIdentifier : BOOL
VAR_INPUT
	Identifier : T_MAXSTRING;
	Destination : REFERENCE TO I_StructuredDatatype;
END_VAR
TryGetStructureByIdentifier := structures.TryGetValue(Identifier, Destination);
END_METHOD

END_FUNCTION_BLOCK

// ---- mobject-events/EventEmitter/EventEmitter.TcPOU
{attribute 'linkalways'} 
{attribute 'no_explicit_call' := 'This FB is a CLASS and must be accessed using methods or properties'}
{attribute 'enable_dynamic_creation'}
FUNCTION_BLOCK EventEmitter EXTENDS Disposable IMPLEMENTS I_EventEmitter, I_EventTarget
VAR
	firstEventHandlerItem : I_EventHandlerItem;
END_VAR

METHOD PUBLIC Clear
VAR_INPUT
END_VAR
DisposeAllEventHandlerItems();
END_METHOD

METHOD PRIVATE DisposeAllEventHandlerItems
VAR_INPUT
END_VAR
WHILE firstEventHandlerItem <> 0 DO
	DisposeEventHandlerItem(firstEventHandlerItem);
END_WHILE
END_METHOD

METHOD PRIVATE DisposeEventHandlerItem
VAR_INPUT
	EventHandlerItem : I_EventHandlerItem;
END_VAR
RemoveEventHandlerItemFromCollection(EventHandlerItem);
EventHandlerItem.Dispose();
END_METHOD

METHOD PUBLIC Emit
VAR_INPUT
	EventName : T_MaxString;
	Event : I_Event;
END_VAR
VAR
	currentEventHandlerItem : I_EventHandlerItem;
END_VAR
currentEventHandlerItem := firstEventHandlerItem;

WHILE currentEventHandlerItem <> 0 DO
	currentEventHandlerItem.Emit(EventName, Event);
	currentEventHandlerItem := currentEventHandlerItem.Next;
END_WHILE
END_METHOD

METHOD FB_exit : BOOL
VAR_INPUT
	bInCopyCode : BOOL; // if TRUE, the exit method is called for exiting an instance that is copied afterwards (online change).
END_VAR
IF bInCopyCode THEN
	RETURN;
END_IF

DisposeAllEventHandlerItems();
END_METHOD

METHOD PRIVATE FindEventHandlerItem : I_EventHandlerItem
VAR_INPUT
	EventName : T_MaxString;
	EventHandler : I_EventHandler;
END_VAR
VAR
	currentEventHandlerItem : I_EventHandlerItem;
END_VAR
currentEventHandlerItem := firstEventHandlerItem;

WHILE currentEventHandlerItem <> 0 DO
	
	IF currentEventHandlerItem.EqualTo(EventName, EventHandler) THEN
		FindEventHandlerItem := currentEventHandlerItem; 
		RETURN;
	END_IF
	
	currentEventHandlerItem := currentEventHandlerItem.Next;

END_WHILE
END_METHOD

METHOD PRIVATE InsertEventHandlerItem
VAR_INPUT
	EventHandlerItem : I_EventHandlerItem;
END_VAR
VAR
	currentEventHandlerItem : I_EventHandlerItem;
END_VAR
IF firstEventHandlerItem = 0 THEN
	firstEventHandlerItem := EventHandlerItem;
	RETURN;
END_IF

currentEventHandlerItem := firstEventHandlerItem;

WHILE currentEventHandlerItem.next <> 0 DO
	currentEventHandlerItem := currentEventHandlerItem.next;
END_WHILE

currentEventHandlerItem.next := EventHandlerItem;
EventHandlerItem.previous := currentEventHandlerItem;
END_METHOD

METHOD PUBLIC OffEvent
VAR_INPUT
	EventName : T_MaxString;
	EventHandler : I_EventHandler;
END_VAR
VAR
	foundHandlerItem : I_EventHandlerItem;
END_VAR
foundHandlerItem := FindEventHandlerItem(EventName, EventHandler);

IF foundHandlerItem = 0 THEN
	RETURN;
END_IF

DisposeEventHandlerItem(foundHandlerItem);
END_METHOD

METHOD PUBLIC OnceEvent
VAR_INPUT
	EventName : T_MaxString;
	EventHandler : I_EventHandler;
END_VAR
VAR
	pEventHandlerItem : POINTER TO EventHandlerItemOnceOnly;
END_VAR
pEventHandlerItem := __NEW(EventHandlerItemOnceOnly(Name := EventName, Handler := EventHandler, Parent := THIS^));
InsertEventHandlerItem(pEventHandlerItem^);
END_METHOD

METHOD PUBLIC OnEvent
VAR_INPUT
	EventName : T_MaxString;
	EventHandler : I_EventHandler;
END_VAR
VAR
	pEventHandlerItem : POINTER TO EventHandlerItem;
END_VAR
pEventHandlerItem := __NEW(EventHandlerItem(Name :=EventName, Handler := EventHandler));
InsertEventHandlerItem(pEventHandlerItem^);
END_METHOD

METHOD PRIVATE RemoveEventHandlerItemFromCollection
VAR_INPUT
	EventHandlerItem : I_EventHandlerItem;
END_VAR
VAR
	previous : I_EventHandlerItem;
	next : I_EventHandlerItem;
END_VAR
IF EventHandlerItem = 0 THEN
	// nothing to remove
	RETURN;
END_IF

IF EventHandlerItem = firstEventHandlerItem AND EventHandlerItem.Next = 0 THEN 
	
	// the item was the only one in the list, as such you just set the first to zero
	firstEventHandlerItem := 0; 
	
ELSIF EventHandlerItem = firstEventHandlerItem THEN 
	
	// the item was the first in the list of many, so make the next item the first and remove 
	// it's "previous" as the first in the item does not have a previous
	firstEventHandlerItem := EventHandlerItem.next; 
	firstEventHandlerItem.Previous := 0;

ELSIF EventHandlerItem.Next <> 0 THEN
	
	// the item is mid list so link it's previous and next together 
	previous := EventHandlerItem.Previous;
	next := EventHandlerItem.Next;
	
	previous.Next := next;
	next.Previous := previous;
	
ELSE 
	
	// the item is at the end so only remove itself from the previous
	previous := EventHandlerItem.Previous;
	previous.Next := 0;

END_IF
END_METHOD

END_FUNCTION_BLOCK

// ---- mobject-events/_Internal/EventHandlerItem/EventHandlerItem.TcPOU
{attribute 'linkalways'} 
{attribute 'no_explicit_call' := 'This FB is a CLASS and must be accessed using methods or properties'}
{attribute 'enable_dynamic_creation'}
FUNCTION_BLOCK EventHandlerItem EXTENDS Disposable IMPLEMENTS I_EventHandlerItem
VAR
	name : T_MAXSTRING;
	handler : I_EventHandler;
	_next : I_EventHandlerItem;
	_previous : I_EventHandlerItem;
END_VAR

METHOD PUBLIC Emit
VAR_INPUT
	EventName : T_MaxString;
	Event : I_Event;
END_VAR
IF EventName <> name THEN
	RETURN;
END_IF

IF handler = 0 THEN
	RETURN;
END_IF

handler.HandleEvent(Event);
END_METHOD

METHOD PUBLIC EqualTo : BOOL
VAR_INPUT
	Name : T_MaxString;
	Handler : I_EventHandler;
END_VAR
IF THIS^.handler <> Handler THEN
	RETURN;
END_IF

IF THIS^.name <> Name THEN
	RETURN;
END_IF

EqualTo := TRUE;
END_METHOD

METHOD FB_init : BOOL
VAR_INPUT
	bInitRetains : BOOL; // if TRUE, the retain variables are initialized (warm start / cold start)
	bInCopyCode : BOOL;  // if TRUE, the instance afterwards gets moved into the copy code (online change)
	Name : T_MAXSTRING;
	Handler : I_EventHandler;
END_VAR
THIS^.name := Name;
THIS^.handler := Handler;
END_METHOD

PROPERTY PUBLIC Next : I_EventHandlerItem
GET
Next := _next;
END_GET
SET
_next := Next;
END_SET
END_PROPERTY

PROPERTY PUBLIC Previous : I_EventHandlerItem
GET
Previous := _previous;
END_GET
SET
_previous := Previous;
END_SET
END_PROPERTY

END_FUNCTION_BLOCK

// ---- mobject-collections/Dictionary/Dictionary.TcPOU
{attribute 'linkalways'} 
{attribute 'no_explicit_call' := 'This FB is a CLASS and must be accessed using methods or properties'}
{attribute 'enable_dynamic_creation'}
FUNCTION_BLOCK Dictionary EXTENDS Disposable IMPLEMENTS I_Dictionary
VAR
	eventEmitter : EventEmitter;
	rootNode : I_DictionaryTreeNode;
END_VAR

METHOD PUBLIC AddOrUpdate
VAR_INPUT
	Key : T_MAXSTRING;
	Value : ANY;
END_VAR
rootNode := THIS^.RecursiveInsert(Key, Value, rootNode);
EmitChangedEvent();
END_METHOD

METHOD PRIVATE Balance : I_DictionaryTreeNode
VAR_INPUT
	Node : I_DictionaryTreeNode;
END_VAR
VAR
	balanceFactor : DINT;
END_VAR
balanceFactor := THIS^.GetBalanceFactor(Node);

IF (balanceFactor > 1) THEN
	IF THIS^.GetBalanceFactor(Node.Left) < 0 THEN
		Node.Left := THIS^.LeftRotate(Node.Left);
	END_IF
	Node := RightRotate(Node);
ELSIF (balanceFactor < -1) THEN
	IF THIS^.GetBalanceFactor(Node.Right) > 0 THEN
		Node.Right := RightRotate(Node.Right);
	END_IF
	Node := LeftRotate(Node);
END_IF

Balance := Node;
END_METHOD

METHOD PUBLIC Clear
VAR_INPUT
END_VAR
IF rootNode = 0 THEN
	RETURN;
END_IF

THIS^.RecursiveClear(rootNode);
rootNode := 0;
EmitChangedEvent();
END_METHOD

METHOD PUBLIC ContainsKey : BOOL
VAR_INPUT
	Key : T_MAXSTRING;
END_VAR
VAR
	foundNode : I_DictionaryTreeNode;
END_VAR
foundNode := THIS^.RecursiveFind(Key, rootNode);

IF foundNode = 0 THEN
	RETURN;
END_IF

ContainsKey := TRUE;
END_METHOD

PROPERTY PUBLIC Count : DINT
GET
VAR
	NodeCount : DINT;
END_VAR
RecursiveCountNodes(rootNode, NodeCount);
Count := NodeCount;
END_GET
END_PROPERTY

METHOD PRIVATE EmitChangedEvent
VAR
	pDictionaryChangedEvent : POINTER TO KeyValueCollectionChangedEvent;
END_VAR
pDictionaryChangedEvent := __NEW(KeyValueCollectionChangedEvent(Target := THIS^));
eventEmitter.Emit('OnChanged', pDictionaryChangedEvent^);
pDictionaryChangedEvent^.Dispose();
END_METHOD

METHOD PRIVATE EmitDisposedEvent
VAR
	pDictionaryDisposedEvent : POINTER TO KeyValueCollectionDisposedEvent;
END_VAR
pDictionaryDisposedEvent := __NEW(KeyValueCollectionDisposedEvent(Target := THIS^));
eventEmitter.Emit('OnDisposed', pDictionaryDisposedEvent^);
pDictionaryDisposedEvent^.Dispose();
END_METHOD

METHOD FB_exit : BOOL
VAR_INPUT
	bInCopyCode : BOOL; // if TRUE, the exit method is called for exiting an instance that is copied afterwards (online change).
END_VAR
VAR
END_VAR
IF bInCopyCode THEN
    RETURN;
END_IF

Clear();
EmitDisposedEvent();
END_METHOD

METHOD PRIVATE FindMinimum : I_DictionaryTreeNode
VAR_INPUT
	Node : I_DictionaryTreeNode;
END_VAR
VAR
	nextNode : I_DictionaryTreeNode;
END_VAR
nextNode := Node;

WHILE (nextNode.left <> 0) DO
      nextNode := nextNode.left;
END_WHILE;

FindMinimum := nextNode;
END_METHOD

METHOD PRIVATE GetBalanceFactor : DINT
VAR_INPUT
	Node : I_DictionaryTreeNode;
END_VAR
IF (Node = 0) THEN
	GetBalanceFactor := 0;
	RETURN;
END_IF

GetBalanceFactor := THIS^.GetHeight(node.left) - THIS^.GetHeight(node.right);
END_METHOD

METHOD GetEnumerator : I_ForwardEnumerator
VAR
	pNodeCollection : POINTER TO LinkedList;
	pEnumerator : POINTER TO DictionaryForwardEnumerator;
END_VAR
pNodeCollection := __NEW(LinkedList);
THIS^.RecursiveAddNodesInOrderToCollection(rootNode, pNodeCollection^);

pEnumerator := __NEW(DictionaryForwardEnumerator(Parent := THIS^, Nodes := pNodeCollection^));
GetEnumerator := pEnumerator^;
END_METHOD

METHOD PRIVATE GetHeight : DINT
VAR_INPUT
	Node : I_DictionaryTreeNode;
END_VAR
IF Node = 0 THEN
	GetHeight := -1;
	RETURN;
END_IF

GetHeight := Node.Height;
END_METHOD

METHOD PUBLIC GetKeys : I_Collection
VAR
	pLinkedList : POINTER TO LinkedList;
END_VAR
pLinkedList := __NEW(LinkedList);
THIS^.RecursiveAddKeysInOrderToCollection(rootNode,pLinkedList^);
GetKeys := pLinkedList^;
END_METHOD

METHOD GetKeyValueEnumerator : I_KeyValueForwardEnumerator
VAR
	pNodeCollection : POINTER TO LinkedList;
	pEnumerator : POINTER TO DictionaryForwardEnumerator;
END_VAR
pNodeCollection := __NEW(LinkedList);
THIS^.RecursiveAddNodesInOrderToCollection(rootNode, pNodeCollection^);

pEnumerator := __NEW(DictionaryForwardEnumerator(Parent := THIS^, Nodes := pNodeCollection^));
GetKeyValueEnumerator := pEnumerator^;
END_METHOD

PROPERTY IsEmpty : BOOL
GET
IsEmpty := rootNode = 0;
END_GET
END_PROPERTY

METHOD PRIVATE LeftRotate : I_DictionaryTreeNode
VAR_INPUT
	X : I_DictionaryTreeNode;
END_VAR
VAR
	y : I_DictionaryTreeNode;
	t2 : I_DictionaryTreeNode;
END_VAR
y := X.right;
t2 := y.left;
y.left := X;
X.right := t2;
THIS^.UpdateHeight(X);
THIS^.UpdateHeight(y);
LeftRotate := y;
END_METHOD

METHOD PUBLIC OffEvent
VAR_INPUT
	EventName : T_MaxString;
	EventHandler : I_EventHandler;
END_VAR
eventEmitter.OffEvent(EventName, EventHandler);
END_METHOD

METHOD PUBLIC OnceEvent
VAR_INPUT
	EventName : T_MaxString;
	EventHandler : I_EventHandler;
END_VAR
eventEmitter.OnceEvent(EventName, EventHandler);
END_METHOD

METHOD PUBLIC OnEvent
VAR_INPUT
	EventName : T_MaxString;
	EventHandler : I_EventHandler;
END_VAR
eventEmitter.OnEvent(EventName, EventHandler);
END_METHOD

METHOD PRIVATE RecursiveAddKeysInOrderToCollection
VAR_INPUT
	Node : I_DictionaryTreeNode;
	Collection : I_Collection;
END_VAR
VAR
	key : T_MAXSTRING;
END_VAR
IF Node = 0 THEN
	RETURN;
END_IF

THIS^.RecursiveAddKeysInOrderToCollection(Node.Left,Collection);
key := Node.Key;
Collection.AddItem(key);
THIS^.RecursiveAddKeysInOrderToCollection(Node.Right,Collection);
END_METHOD

METHOD PRIVATE RecursiveAddNodesInOrderToCollection
VAR_INPUT
	Node : I_DictionaryTreeNode;
	Collection : I_Collection;
END_VAR
IF Node = 0 THEN
	RETURN;
END_IF

THIS^.RecursiveAddNodesInOrderToCollection(Node.Left,Collection);
Collection.AddItem(Node);
THIS^.RecursiveAddNodesInOrderToCollection(Node.Right,Collection);
END_METHOD

METHOD PRIVATE RecursiveClear
VAR_INPUT
	Node : I_DictionaryTreeNode;
END_VAR
VAR
	thisNodeKey : T_MAXSTRING;
	leftNodeKey : T_MAXSTRING;
	rightNodeKey : T_MAXSTRING;
END_VAR
IF (Node = 0) THEN
	RETURN;
END_IF

thisNodeKey := Node.key;

IF (Node.Left <> 0) THEN
	leftNodeKey := Node.Left.key;
END_IF

IF (Node.Right <> 0) THEN
	rightNodeKey := Node.Right.key;
END_IF


RecursiveClear(Node.Left);
RecursiveClear(Node.Right);
Node.Dispose();
END_METHOD

METHOD PRIVATE RecursiveCountNodes
VAR_INPUT
	Node : I_DictionaryTreeNode;
	Count : REFERENCE TO DINT;
END_VAR
IF Node = 0 THEN
	RETURN;
END_IF

Count := Count + 1;

THIS^.RecursiveCountNodes(Node.Left,Count);
THIS^.RecursiveCountNodes(Node.Right,Count);
END_METHOD

METHOD PRIVATE RecursiveDelete : I_DictionaryTreeNode
VAR_INPUT
	Key : T_MAXSTRING;
	Node : I_DictionaryTreeNode;
END_VAR
VAR
	newNode : I_DictionaryTreeNode; 
	minValueNode : I_DictionaryTreeNode;
	minValueNodeParent : I_DictionaryTreeNode;
	balanceFactor : DINT;
END_VAR
IF (Node = 0) THEN
    RETURN;
END_IF

IF (Key < Node.Key) THEN
    Node.left := THIS^.RecursiveDelete(Key, Node.left);
ELSIF (Key > Node.Key) THEN
    Node.right := THIS^.RecursiveDelete(Key, Node.right);
ELSE
    IF (Node.Left = 0) OR (Node.Right = 0) THEN
        IF (Node.Left = 0) THEN
            newNode := Node.Right;
        ELSE
            newNode := Node.Left;
        END_IF

        Node.Dispose();
        THIS^.updateHeight(newNode);
        RecursiveDelete := THIS^.Balance(newNode);
        RETURN;
    ELSE
        minValueNode := FindMinimum(Node.Right);
        Node.Clone(minValueNode);
        Node.Right := THIS^.RecursiveDelete(minValueNode.Key, Node.Right);	
    END_IF
END_IF

THIS^.updateHeight(Node);
RecursiveDelete := THIS^.Balance(Node);
END_METHOD

METHOD PRIVATE RecursiveFind : I_DictionaryTreeNode
VAR_INPUT
	Key : T_MAXSTRING;
	Node : I_DictionaryTreeNode;
END_VAR
IF (Node = 0) THEN
	RETURN;
END_IF

IF (Key < Node.key) THEN
  RecursiveFind := THIS^.RecursiveFind(key, Node.left);
  RETURN;
ELSIF (key > Node.key) THEN
  RecursiveFind := THIS^.RecursiveFind(key, Node.right);
  RETURN;
ELSE 
  RecursiveFind := Node;
  RETURN;
END_IF
END_METHOD

METHOD PRIVATE RecursiveInsert : I_DictionaryTreeNode
VAR_INPUT
	Key : T_MAXSTRING;
	Value : ANY;
	Node : I_DictionaryTreeNode;
END_VAR
VAR
	pAVLTreeNode : POINTER TO DictionaryTreeNode;
	balanceFactor : DINT;
END_VAR
IF (Node = 0) THEN
	pAVLTreeNode := __NEW(DictionaryTreeNode(NodeKey := Key, NodeSource := Value));
	RecursiveInsert := pAVLTreeNode^;
	RETURN;
END_IF

IF (Key < Node.Key) THEN
	Node.left := THIS^.RecursiveInsert(Key, Value, Node.left);
ELSIF (Key > Node.Key) THEN
	Node.right := THIS^.RecursiveInsert(Key, Value, Node.right);
ELSE
	Node.Reinitialize(Key,Value);
	RecursiveInsert := Node;
END_IF

THIS^.updateHeight(node);

balanceFactor := THIS^.GetBalanceFactor(Node);
Node := balance(Node);
RecursiveInsert := Node;
END_METHOD

METHOD PUBLIC Remove
VAR_INPUT
	Key : T_MAXSTRING;
END_VAR
rootNode := THIS^.RecursiveDelete(Key, rootNode);
EmitChangedEvent();
END_METHOD

METHOD PRIVATE RightRotate : I_DictionaryTreeNode
VAR_INPUT
	Y : I_DictionaryTreeNode;
END_VAR
VAR
	x : I_DictionaryTreeNode;
	t2 : I_DictionaryTreeNode;
END_VAR
x := Y.left;
t2 := x.right;
x.right := Y;
Y.left := t2;
THIS^.UpdateHeight(Y);
THIS^.UpdateHeight(x);
RightRotate := x;
END_METHOD

METHOD PUBLIC TryAdd : BOOL
VAR_INPUT
	Key : T_MAXSTRING;
	Value : ANY;
END_VAR
IF ContainsKey(Key) THEN
	RETURN;
END_IF
	  
THIS^.AddOrUpdate(Key, Value);
TryAdd := TRUE;
END_METHOD

METHOD PUBLIC TryGetValue : BOOL
VAR_INPUT
	Key : T_MAXSTRING;
	Destination	: ANY;
END_VAR
TryGetValue := TryGetValueTo(Key, Destination.pValue, DINT_TO_UDINT(Destination.diSize));
END_METHOD

METHOD PUBLIC TryGetValueTo : BOOL
VAR_INPUT
	Key : T_MAXSTRING;
	DestinationAddress : PVOID;
	DestinationSize : UDINT;
END_VAR
VAR
	foundNode : I_DictionaryTreeNode;
END_VAR
foundNode := THIS^.RecursiveFind(Key, rootNode);

IF foundNode = 0 THEN
	RETURN;
END_IF

TryGetValueTo := foundNode.TryGetTo(DestinationAddress, DestinationSize);
END_METHOD

METHOD PRIVATE UpdateHeight
VAR_INPUT
	Node : I_DictionaryTreeNode;
END_VAR
IF (Node = 0) THEN
	RETURN;
END_IF

Node.height := 1 + MAX(THIS^.GetHeight(Node.left), THIS^.GetHeight(Node.right));
END_METHOD

END_FUNCTION_BLOCK

// ---- mobject-collections/_Internal/Events/KeyValueCollection/KeyValueCollectionChangedEvent.TcPOU
{attribute 'linkalways'} 
{attribute 'no_explicit_call' := 'This FB is a CLASS and must be accessed using methods or properties'}
{attribute 'enable_dynamic_creation'}
FUNCTION_BLOCK KeyValueCollectionChangedEvent EXTENDS KeyValueCollectionEvent IMPLEMENTS I_KeyValueCollectionChangedEvent

END_FUNCTION_BLOCK

// ---- mobject-collections/_Internal/Events/KeyValueCollection/KeyValueCollectionEvent.TcPOU
{attribute 'linkalways'} 
{attribute 'no_explicit_call' := 'This FB is a CLASS and must be accessed using methods or properties'}
{attribute 'enable_dynamic_creation'}
FUNCTION_BLOCK ABSTRACT KeyValueCollectionEvent EXTENDS Disposable
VAR
	_target : I_KeyValueCollection;
END_VAR

METHOD FB_init : BOOL
VAR_INPUT
	bInitRetains : BOOL; // if TRUE, the retain variables are initialized (warm start / cold start)
	bInCopyCode : BOOL;  // if TRUE, the instance afterwards gets moved into the copy code (online change)
	Target : I_KeyValueCollection;
END_VAR
This^._target := Target;
END_METHOD

PROPERTY PUBLIC Target : I_KeyValueCollection
GET // PUBLIC
Target := _target;
END_GET
END_PROPERTY

END_FUNCTION_BLOCK

// ---- mobject-collections/_Internal/Events/KeyValueCollection/KeyValueCollectionDisposedEvent.TcPOU
{attribute 'linkalways'} 
{attribute 'no_explicit_call' := 'This FB is a CLASS and must be accessed using methods or properties'}
{attribute 'enable_dynamic_creation'}
FUNCTION_BLOCK KeyValueCollectionDisposedEvent EXTENDS KeyValueCollectionEvent IMPLEMENTS I_KeyValueCollectionDisposedEvent

END_FUNCTION_BLOCK

// ---- mobject-collections/LinkedList/LinkedList.TcPOU
{attribute 'linkalways'} 
{attribute 'no_explicit_call' := 'This FB is a CLASS and must be accessed using methods or properties'}
{attribute 'enable_dynamic_creation'}
FUNCTION_BLOCK LinkedList EXTENDS Disposable IMPLEMENTS I_LinkedList
VAR
	head : I_LinkedListNode;
	tail : I_LinkedListNode;
	eventEmitter : EventEmitter;
END_VAR

METHOD PUBLIC AddAfter
VAR_INPUT
	After : I_LinkedListNode;
	Value : ANY;
END_VAR
VAR
	node : I_LinkedListNode;
END_VAR
IF NOT ContainsLinkedListNode(After) THEN
	RETURN;
END_IF

node := CreateNode(Value);
AddNodeAfter(After,node);
EmitChangedEvent();
END_METHOD

METHOD PUBLIC AddBefore
VAR_INPUT
	Before : I_LinkedListNode;
	Value : ANY;
END_VAR
VAR
	node : I_LinkedListNode;
END_VAR
IF NOT ContainsLinkedListNode(Before) THEN
	RETURN;
END_IF

node := CreateNode(Value);
AddNodeBefore(Before,node);
EmitChangedEvent();
END_METHOD

METHOD PUBLIC AddFirst
VAR_INPUT
	Value : ANY;
END_VAR
VAR
	node : I_LinkedListNode;
END_VAR
node := CreateNode(Value);
AddNodeFirst(node);
EmitChangedEvent();
END_METHOD

METHOD PUBLIC AddItem
VAR_INPUT
	Item : ANY;
END_VAR
AddLast(Item);
END_METHOD

METHOD PUBLIC AddLast
VAR_INPUT
	Value : ANY;
END_VAR
VAR
	node : I_LinkedListNode;
END_VAR
node := CreateNode(Value);
AddNodeLast(node);
EmitChangedEvent();
END_METHOD

METHOD PRIVATE AddNodeAfter
VAR_INPUT
	After : I_LinkedListNode;
	Node : I_LinkedListNode;
END_VAR
VAR
	originalNext : I_LinkedListNode;
END_VAR
IF After = tail THEN
	AddNodeLast(Node);
	RETURN;
END_IF

originalNext := After.Next;
After.Next := Node;
Node.Previous := After;
Node.Next := originalNext;
originalNext.Previous := Node;
END_METHOD

METHOD PRIVATE AddNodeBefore
VAR_INPUT
	Before : I_LinkedListNode;
	Node : I_LinkedListNode;
END_VAR
VAR
	originalBefore : I_LinkedListNode;
END_VAR
IF Before = head THEN
	AddNodeFirst(Node);
	RETURN;
END_IF

originalBefore := Before.Previous;
Before.Previous := Node;
Node.Next := Before;
Node.Previous := originalBefore;
originalBefore.Next := Node;
END_METHOD

METHOD PRIVATE AddNodeFirst
VAR_INPUT
	Node : I_LinkedListNode;
END_VAR
VAR
	originalFirst : I_LinkedListNode;
END_VAR
IF IsEmpty THEN
	head := Node;
	tail := Node; 
	RETURN;	
END_IF

originalFirst := head;
head := Node;
Node.Next := originalFirst;
originalFirst.Previous := Node;
END_METHOD

METHOD PRIVATE AddNodeLast
VAR_INPUT
	Node : I_LinkedListNode;
END_VAR
VAR
	originalLast : I_LinkedListNode;
END_VAR
IF IsEmpty THEN
	head := Node;
	tail := Node; 
	RETURN;	
END_IF

originalLast := tail;
tail := Node;
Node.Previous := originalLast;
originalLast.Next := Node;
END_METHOD

METHOD PUBLIC Clear
IF IsEmpty THEN
	return;
END_IF

RemoveAllNodes();
EmitChangedEvent();
END_METHOD

METHOD PUBLIC Contains : BOOL
VAR_INPUT
    Item : ANY;
END_VAR
VAR
    found : I_LinkedListNode;
END_VAR
found := Find(Item);
Contains := found <> 0;
END_METHOD

METHOD PRIVATE ContainsLinkedListNode : BOOL
VAR_INPUT
    Node : I_LinkedListNode;
END_VAR
VAR
	current : I_LinkedListNode;
END_VAR
IF IsEmpty THEN	
	RETURN;
END_IF

current := head; 

WHILE current <> 0 DO
	IF current = Node THEN
		ContainsLinkedListNode := TRUE;
		RETURN;
	END_IF
	current := current.next; 
END_WHILE;
END_METHOD

PROPERTY PUBLIC Count : DINT
GET
VAR
	current : I_LinkedListNode;
END_VAR
current := First;

WHILE current <> 0 DO
	Count := Count + 1;
	current := current.Next;
END_WHILE
END_GET
END_PROPERTY

METHOD PRIVATE CreateNode : I_LinkedListNode
VAR_INPUT
	Value : ANY;
END_VAR
VAR
	pLinkedListItem : POINTER TO LinkedListNode;
END_VAR
pLinkedListItem := __NEW(LinkedListNode(Source := Value)); 
CreateNode := pLinkedListItem^;
END_METHOD

METHOD PRIVATE EmitChangedEvent
VAR
	pCollectionChangedEvent : POINTER TO CollectionChangedEvent;
END_VAR
pCollectionChangedEvent := __NEW(CollectionChangedEvent(Target := THIS^));
eventEmitter.Emit('OnChanged', pCollectionChangedEvent^);
pCollectionChangedEvent^.Dispose();
END_METHOD

METHOD PRIVATE EmitDisposedEvent
VAR
	pCollectionDisposedEvent : POINTER TO CollectionDisposedEvent;
END_VAR
pCollectionDisposedEvent := __NEW(CollectionDisposedEvent(Target := THIS^));
eventEmitter.Emit('OnDisposed', pCollectionDisposedEvent^);
pCollectionDisposedEvent^.Dispose();
END_METHOD

METHOD FB_exit : BOOL
VAR_INPUT
	bInCopyCode : BOOL; // if TRUE, the exit method is called for exiting an instance that is copied afterwards (online change).
END_VAR
IF bInCopyCode THEN
	RETURN;
END_IF

Clear();
EmitDisposedEvent();
END_METHOD

METHOD PUBLIC Find : I_LinkedListNode
VAR_INPUT
	Value : ANY;
END_VAR
Find := FindFirstNodeWithValue(Value);
END_METHOD

METHOD PRIVATE FindFirstNodeWithValue : I_LinkedListNode
VAR_INPUT
	Value : ANY;
END_VAR
VAR
	current : I_LinkedListNode;
END_VAR
IF IsEmpty THEN	
	RETURN;
END_IF

current := head; 

WHILE current <> 0 DO
	IF current.Equals(Value) THEN
		FindFirstNodeWithValue := current;
		RETURN;
	END_IF
	current := current.next; 
END_WHILE;
END_METHOD

METHOD PUBLIC FindLast : I_LinkedListNode
VAR_INPUT
	Value : ANY;
END_VAR
FindLast := FindLastNodeWithValue(Value);
END_METHOD

METHOD PRIVATE FindLastNodeWithValue : I_LinkedListNode
VAR_INPUT
	Value : ANY;
END_VAR
VAR
	current : I_LinkedListNode;
END_VAR
IF IsEmpty THEN	
	RETURN;
END_IF

current := tail; 

WHILE current <> 0 DO
	IF current.Equals(Value) THEN
		FindLastNodeWithValue := current;
		RETURN;
	END_IF
	current := current.Previous; 
END_WHILE;
END_METHOD

PROPERTY PUBLIC First : I_LinkedListNode
GET
First := head;
END_GET
END_PROPERTY

METHOD PUBLIC GetEnumerator : I_ForwardEnumerator
VAR
	pLinkedListForwardEnumerator : POINTER TO LinkedListForwardEnumerator;
END_VAR
pLinkedListForwardEnumerator := __NEW(LinkedListForwardEnumerator(Parent := THIS^));
GetEnumerator := pLinkedListForwardEnumerator^;
END_METHOD

PROPERTY IsEmpty : BOOL
GET
IsEmpty := head = 0;
END_GET
END_PROPERTY

PROPERTY PUBLIC Last : I_LinkedListNode
GET
Last := tail;
END_GET
END_PROPERTY

METHOD PUBLIC OffEvent
VAR_INPUT
	EventName : T_MaxString;
	EventHandler : I_EventHandler;
END_VAR
eventEmitter.OffEvent(EventName, EventHandler);
END_METHOD

